// TIA Portal V19 program export: 5 tag tables, 0 data types, 1 data blocks, 10 code blocks (in call order from the OBs), 0 instance data blocks

VAR_GLOBAL   // PLC tag table "Default tag table"
   memSensorType2 AT %MW14 : Int;
   memSensorType1 AT %MW16 : Int;
   Tag_1 AT %T5 : Timer;
END_VAR
VAR_GLOBAL CONSTANT   // user constants
   PANELS_NO : Int := 2;
   LACYCCOM_BUFFER_ELEMENTS_UPPER_LIM : Int := 59;   // Upper limit of request buffer array
   LACYCCOM_WRITE_PARAMETERS_UPPER_LIM : Int := 18;   // Upper limit of write parameters
   LACYCCOM_READ_PARAMETERS_UPPER_LIM : Int := 38;   // Upper limit of read parameters
   LACYCCOM_SILENT_OPERATION_PARAMETERS_UPPER_LIM : Int := 17;   // Upper limit of parameters in LAcycCom_typeDriveSilentOperation
   LACYCCOM_NO_COMMAND : Byte := 16#00;   // No command
   LACYCCOM_READ_COMMAND : Byte := 16#01;   // Read command
   LACYCCOM_WRITE_COMMAND : Byte := 16#02;   // Write command
   LACYCCOM_TYPE_ALARM : SInt := 1;   // Alarm
   LACYCCOM_TYPE_FAULT : SInt := 2;   // Fault
   LACYCCOM_TYPE_SI_MESSAGE : SInt := 3;   // SI message
   LACYCCOM_MESSAGES_UPPER_LIM : Int := 23;   // Upper limit of elements in LAcycCom_typeDriveMessages (fix value)
END_VAR

VAR_GLOBAL   // PLC tag table "tags_IO"
   "866TR2510-S1_Rev" AT %I0.0 : Bool;   // 866TR2510 - Reverse KP-208
   "866TR2510-S1_Fwd" AT %I0.1 : Bool;   // 866TR2510 - Forward KP-208
   "866TR2520-S1_Rev" AT %I0.2 : Bool;   // 866TR2520 - Reverse KP-208
   "866TR2520-S1_Fwd" AT %I0.3 : Bool;   // 866TR2520 - Forward KP-208
   "866TR2530-S1_Rev" AT %I0.4 : Bool;   // 866TR2530 - Reverse KP-208
   "866TR2530-S1_Fwd" AT %I0.5 : Bool;   // 866TR2530 - Forward KP-208
   "866LE2540-S1_Up" AT %I0.6 : Bool;   // 866LE2540 - Cage up
   "866LE2540-S1_Down" AT %I0.7 : Bool;   // 866LE2540 - Cage down
   "866TR2541-S1_Rev" AT %I1.0 : Bool;   // 866TR2541 - Reverse KP-208
   "866TR2541-S1_Fwd" AT %I1.1 : Bool;   // 866TR2541 - Forward KP-208
   "866TR2542-S1_Rev" AT %I1.2 : Bool;   // 866TR2542 - Reverse
   "866TR2542-S1_Fwd" AT %I1.3 : Bool;   // 866TR2542 - Forward
   "866MA2543-S1_In" AT %I1.4 : Bool;   // 866MA2543 - In
   "866MA2543-S1_Out" AT %I1.5 : Bool;   // 866MA2543 - Out
   "866TR2510-GL1" AT %I1.6 : Bool;   // 866TR2510 - Entry photocell
   "866TR2510-GL2" AT %I1.7 : Bool;   // 866TR2510 - Exit photocell
   "866TR2520-GL1" AT %I2.0 : Bool;   // 866TR2520 - Entry photocell
   "866TR2520-GL2" AT %I2.1 : Bool;   // 866TR2520 - Exit photocell
   "866TR2530-GL1" AT %I2.2 : Bool;   // 866TR2530 - Entry photocell
   "866TR2530-GL2" AT %I2.3 : Bool;   // 866TR2530 - Exit photocell
   "2510_KontrollOrd" AT %QW400 : Word;
   "2510_StatusOrd" AT %IW400 : Word;
   "2510_SpeedSP" AT %QW402 : Word;
   "2510_SpeedPV" AT %IW402 : Word;
   "2520_KontrollOrd" AT %QW388 : Word;
   "2520_StatusOrd" AT %IW388 : Word;
   "2520_SpeedSP" AT %QW390 : Word;
   "2520_SpeedPV" AT %IW390 : Word;
   "2530_KontrollOrd" AT %QW376 : Word;
   "2530_StatusOrd" AT %IW376 : Word;
   "2530_SpeedSP" AT %QW378 : Word;
   "2530_SpeedPV" AT %IW378 : Word;
   "2600_KontrollOrd" AT %QW412 : Word;
   "2600_StatusOrd" AT %IW412 : Word;
   "2600_SpeedSP" AT %QW414 : Word;
   "2600_SpeedPV" AT %IW414 : Word;
   "101LT1" AT %IW100 : Word;   // Tank 101 Level transmitter 1
   "101LT2" AT %IW102 : Word;   // Tank 101 Level transmitter 2
   "102LT1" AT %IW104 : Word;   // Tank 102 Level transmitter 1
   "102LT2" AT %IW106 : Word;   // Tank 102 Level transmitter 2
   "101CV1" AT %QW100 : Word;   // Tank 101 Control valve 1
   "101CV2" AT %QW102 : Word;   // Tank 101 Control valve 2
   "102CV1" AT %QW104 : Word;   // Tank 102 Control valve 1
   "102CV2" AT %QW106 : Word;   // Tank 102 Control valve 2
   "101PT1" AT %IW108 : Word;   // Tank 101 Pressure transmitter 1
   "101PT2" AT %IW110 : Word;   // Tank 101 Pressure transmitter 2
   "102PT1" AT %IW112 : Word;   // Tank 102 Pressure transmitter 1
   "102PT2" AT %IW114 : Word;   // Tank 102 Pressure transmitter 2
   "101FT1" AT %IW116 : Word;   // Tank 101 Flow transmitter 1
   "101FT2" AT %IW118 : Word;   // Tank 101 Flow transmitter 2
   "102FT1" AT %IW120 : Word;   // Tank 102 Flow transmitter 1
   "102FT2" AT %IW122 : Word;   // Tank 102 Flow transmitter 2
   "101DV1_GL1" AT %I3.0 : Bool;   // 101DV1 Digital valve open feedback
   "101DV1_GL2" AT %I3.1 : Bool;   // 101DV1 Digital valve closed feedback
   "101DV2_GL1" AT %I3.2 : Bool;   // 101DV2 Digital valve open feedback
   "101DV2_GL2" AT %I3.3 : Bool;   // 101DV2 Digital valve closed feedback
   "101DV1_OPEN" AT %Q0.0 : Bool;
   "101DV2_OPEN" AT %Q0.1 : Bool;
END_VAR

VAR_GLOBAL   // PLC tag table "tags_Omriktare"
   Forward AT %M0.0 : Bool;   // Command
   Backward AT %M0.1 : Bool;   // Command
   Acknowledge AT %M0.2 : Bool;   // Command
   SpeedRequest AT %MW2 : Int;   // Command
   TorqueRequest AT %MW4 : Int;   // Command
   Status AT %MW6 : Word;   // Status
   Speed_CV AT %MW8 : Int;   // Status
   Torque_CV AT %MW10 : Int;   // Status
   Alarm AT %M0.3 : Bool;   // Status
   Alarm_number AT %MW12 : Int;   // Status
END_VAR

VAR_GLOBAL   // PLC tag table "tags_Open Library"
END_VAR
VAR_GLOBAL CONSTANT   // user constants
   "Modes.Auto" : Int := 1;
   "Modes.Manual" : Int := 2;
   "Modes.Independent" : Int := 10;
   "Modes.Stop" : Int := 0;
   "HMI.Status.Stopped" : Int := 0;
   "HMI.Status.Estop" : Int := 1;
   "HMI.Status.Error" : Int := 2;
   "HMI.Status.ForwardWork" : Int := 3;
   "HMI.Status.ReverseHome" : Int := 4;
   "HMI.Status.OnForwardWork" : Int := 5;
   "HMI.Status.OnReverseHome" : Int := 6;
   "IoScaling.S7Analog.Default.iRawMax" : Int := 27648;
   "IoScaling.S7Analog.Default.iRawMin" : Int := 0;
   "IoScaling.S7Analog.Default.bSwapBytes" : Bool := false;
   "IoScaling.S7Analog.+-V/mA.iRawMax" : Int := 27648;
   "IoScaling.S7Analog.+-V/mA.iRawMin" : Int := -27648;
   "IoScaling.S7Analog.Types.Default" : Int := 0;
   "IoScaling.S7Analog.Pt100.iRawMax" : Int := 8500;
   "IoScaling.S7Analog.Pt100.iRawMin" : Int := -2000;
   "IoScaling.S7Analog.Pt100.Climate.iRawMax" : Int := 13000;
   "IoScaling.S7Analog.Pt100.Climate.iRawMin" : Int := -12000;
   "IoScaling.S7Analog.Ni100.iRawMax" : Int := 2500;
   "IoScaling.S7Analog.Ni100.iRawMin" : Int := -600;
   "IoScaling.S7Analog.Ni100.Climate.iRawMax" : Int := 25000;
   "IoScaling.S7Analog.Ni100.Climate.iRawMin" : Int := -6000;
   "IoScaling.S7Analog.Types.+-V/mA" : Int := 1;
   "IoScaling.S7Analog.Types.Pt100" : Int := 2;
   "IoScaling.S7Analog.Types.Pt100.Climate" : Int := 3;
   "IoScaling.S7Analog.Types.Ni100" : Int := 4;
   "IoScaling.S7Analog.Types.Ni100.Climate" : Int := 5;
   "IoScaling.S7Analog.Pt100.rScaledMax" : Real := 850.0;
   "IoScaling.S7Analog.Pt100.rScaledMin" : Real := -200.0;
   "IoScaling.S7Analog.Pt100.Climate.rScaledMax" : Real := 130.0;
   "IoScaling.S7Analog.Pt100.Climate.rScaledMin" : Real := -120.0;
   "IoScaling.S7Analog.Ni100.rScaledMax" : Real := 250.0;
   "IoScaling.S7Analog.Ni100.rScaledMin" : Real := -60.0;
   "IoScaling.S7Analog.Ni100.Climate.rScaledMax" : Real := 250.0;
   "IoScaling.S7Analog.Ni100.Climate.rScaledMin" : Real := -60.0;
   "IoScaling.S7Analog.150Ohms.rScaledMax" : Real := 150.0;
   "IoScaling.S7Analog.150Ohms.rScaledMin" : Real := 0.0;
   "IoScaling.S7Analog.300Ohms.rScaledMax" : Real := 300.0;
   "IoScaling.S7Analog.300Ohms.rScaledMin" : Real := 0.0;
   "IoScaling.S7Analog.600Ohms.rScaledMax" : Real := 600.0;
   "IoScaling.S7Analog.600Ohms.rScaledMin" : Real := 0.0;
   "Estop.MinSetPoint" : Int := 0;
   "Estop.MaxSetPoint" : Int := 1;
   "Estop.HMISetPoint" : Int := 2;
   "Modes.PID.Inactive" : Int := 0;
   "Modes.PID.Pretuning" : Int := 1;
   "Modes.PID.FineTuning" : Int := 2;
   "Modes.PID.AutoMode" : Int := 3;
   "Modes.PID.ManualMode" : Int := 4;
   "HMI.Status.Generic1" : Int := 101;
   "HMI.Status.Generic2" : Int := 102;
   "HMI.Status.Generic3" : Int := 103;
   "HMI.Status.Generic4" : Int := 104;
   "HMI.Status.Generic5" : Int := 105;
   "HMI.Status.GenericNone" : Int := 100;
   "HMI.Status.Generic6" : Int := 106;
   "DataTypes.rMaxReal" : Real := 3.402823e38;
   "DataTypes.rMinReal" : Real := -3.402823e38;
   "DataTypes.iMaxInt" : Int := 32767;
   "DataTypes.iMinInt" : Int := -32768;
   "Handshakes.iSize" : Int := 5;
   "SoftStarter.Types.3RW30" : Int := 30;
   "SoftStarter.Types.3RW40" : Int := 40;
   "Simocode.Types.OverloadRelay" : Int := 0;
   "Simocode.Types.DirectStarter" : Int := 1;
   "Simocode.Types.ReversingStarter" : Int := 2;
   "SoftStarter.HMI.Status.RampDown" : Int := 5;
   "SoftStarter.HMI.Status.On" : Int := 4;
   "SoftStarter.HMI.Status.RampUp" : Int := 3;
   "SoftStarter.HMI.Status.EStop" : Int := 1;
   "SoftStarter.HMI.Status.Off" : Int := 0;
   "SoftStarter.HMI.Status.Error" : Int := 2;
   "FIFO.iQueueSize" : Int := 5;
   "FIFO.iQueueDisabled" : Int := -1;
   "TotalizerTimeUnits.MILLISECONDS" : Int := 0;
   "TotalizerTimeUnits.SECONDS" : Int := 1;
   "TotalizerTimeUnits.MINUTES" : Int := 2;
   "TotalizerTimeUnits.HOURS" : Int := 3;
   "TotalizerTimeUnits.DAYS" : Int := 4;
   "HMI.Status.SimulatedForwardWork" : Int := 7;
   "HMI.Status.SimulatedOnForwardWork" : Int := 9;
   "HMI.Status.SimulatedReverseHome" : Int := 8;
   "HMI.Status.SimulatedOnReverseHome" : Int := 10;
   "Ramp.Continuous" : Int := 0;
   "Ramp.Timed" : Int := 1;
END_VAR

VAR_GLOBAL   // PLC tag table "tags_Testtags"
   V1_Test AT %MD30 : Real;
   V2_Test AT %MD34 : Real;
   T1 AT %M38.0 : Bool;
   T2 AT %M38.1 : Bool;
   T3 AT %M38.2 : Bool;
   T4 AT %M38.3 : Bool;
   T5 AT %M38.4 : Bool;
   TI1 AT %MW40 : Int;
   TI2 AT %MW42 : Int;
   TI3 AT %MW44 : Int;
   TI4 AT %MW46 : Int;
END_VAR

DATA_BLOCK "Interface"   // DB18
{ S7_Optimized_Access := 'TRUE' }
// stored: MemoryReserve 100
   VAR
      LT1_ScaledInput : Real;
      LC1_ControllerOuput : Real;
      LC1_ExtSp : Real := 2.5;
      CV2_ExpSp : Real := 20.0;
      "101CV1_Open" : Bool;
   END_VAR
BEGIN
END_DATA_BLOCK

ORGANIZATION_BLOCK "Drives"   // OB1, FBD, ProgramCycle
TITLE = "Main Program Sweep (Cycle)"
{ S7_Optimized_Access := 'TRUE' }
// stored: SetENOAutomatically false
   VAR_INPUT
      Initial_Call : Bool;   // Initial call of this OB
      Remanence : Bool;   // =True, if remanent data are available
   END_VAR
BEGIN

REGION Network 1: 2510!
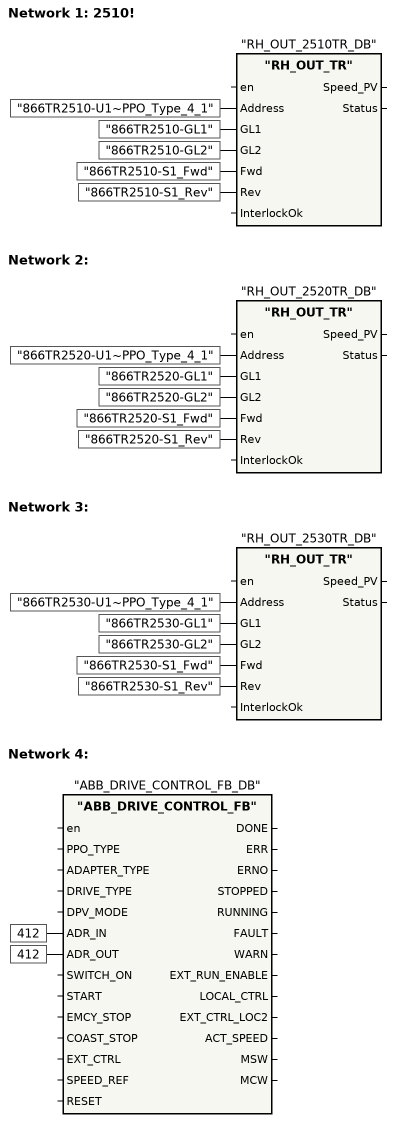
   "RH_OUT_2510TR_DB"(Address := "866TR2510-U1~PPO_Type_4_1",   // "RH_OUT_TR"
                      GL1 := "866TR2510-GL1",
                      GL2 := "866TR2510-GL2",
                      Fwd := "866TR2510-S1_Fwd",
                      Rev := "866TR2510-S1_Rev");
END_REGION

REGION Network 2
   "RH_OUT_2520TR_DB"(Address := "866TR2520-U1~PPO_Type_4_1",   // "RH_OUT_TR"
                      GL1 := "866TR2520-GL1",
                      GL2 := "866TR2520-GL2",
                      Fwd := "866TR2520-S1_Fwd",
                      Rev := "866TR2520-S1_Rev");
END_REGION

REGION Network 3
   "RH_OUT_2530TR_DB"(Address := "866TR2530-U1~PPO_Type_4_1",   // "RH_OUT_TR"
                      GL1 := "866TR2530-GL1",
                      GL2 := "866TR2530-GL2",
                      Fwd := "866TR2530-S1_Fwd",
                      Rev := "866TR2530-S1_Rev");
END_REGION

REGION Network 4
   "ABB_DRIVE_CONTROL_FB_DB"(ADR_IN := 412, ADR_OUT := 412);   // "ABB_DRIVE_CONTROL_FB"
END_REGION
END_ORGANIZATION_BLOCK

FUNCTION_BLOCK "RH_OUT_TR"   // FB1, FBD
{ S7_Optimized_Access := 'TRUE' }
// stored: MemoryReserve 100, SetENOAutomatically false
   VAR_INPUT
      Address : HW_IO;
      GL1 : Bool;
      GL2 : Bool;
      Fwd : Bool;
      Rev : Bool;
      InterlockOk : Bool;
   END_VAR
   VAR_OUTPUT
      Speed_PV : Int;
      Status : Int;
   END_VAR
   VAR
      Frq : "RMP_BIF_FRQ_SPD";   // Device frequency converter control / Laitteen taajuusmuuttajan ohjaus
      Drive { S7_SetPoint := 'True'} : "RMP_FRQ_SPD";
      Control : "RMP_UDT_CONTROL";   // Laitteen ohjaus / Device control
      "Status.Ack" { S7_SetPoint := 'True'} : Bool;
   END_VAR
BEGIN

REGION Network 1: Device fwd request
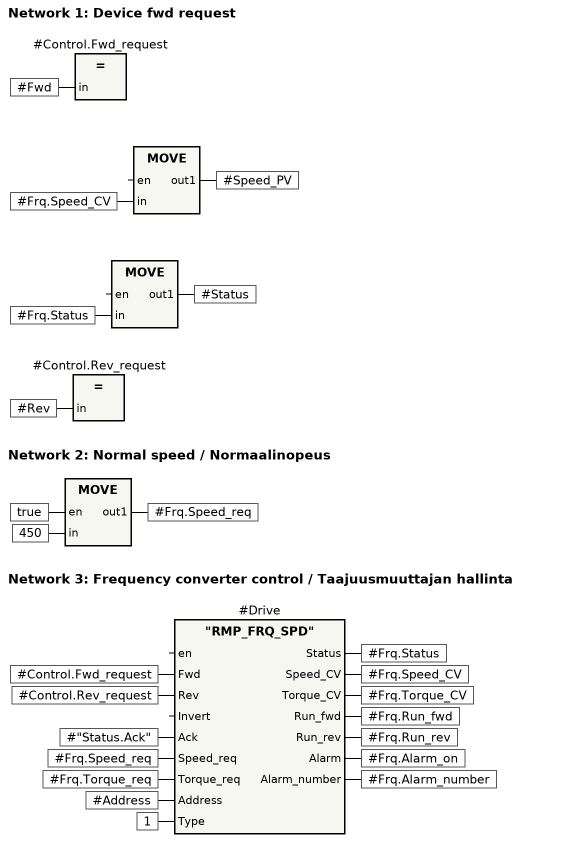
   #Control.Fwd_request := #Fwd;
   #Speed_PV := #Frq.Speed_CV;
   #Status := #Frq.Status;
   #Control.Rev_request := #Rev;
END_REGION

REGION Network 2: Normal speed / Normaalinopeus
   IF true THEN #Frq.Speed_req := 450; END_IF;
END_REGION

REGION Network 3: Frequency converter control / Taajuusmuuttajan hallinta
   #Drive(Fwd := #Control.Fwd_request,   // "RMP_FRQ_SPD"
          Rev := #Control.Rev_request,
          Ack := #"Status.Ack",
          Speed_req := #Frq.Speed_req,
          Torque_req := #Frq.Torque_req,
          Address := #Address,
          "Type" := 1,
          Status => #Frq.Status,
          Speed_CV => #Frq.Speed_CV,
          Torque_CV => #Frq.Torque_CV,
          Run_fwd => #Frq.Run_fwd,
          Run_rev => #Frq.Run_rev,
          Alarm => #Frq.Alarm_on,
          Alarm_number => #Frq.Alarm_number);
END_REGION
END_FUNCTION_BLOCK

FUNCTION_BLOCK "RMP_FRQ_SPD"   // FB11, LAD
TITLE = RMP Sinamics speed & torque control
{ S7_Optimized_Access := 'TRUE' }
AUTHOR : Joni_Lahtonen
FAMILY : Raumaster_Paper
VERSION : 1.0
// This block uses profidrive profile to control siemens frequency converters.
// Use communication profile 352 (6/6) in HW configuration.
// stored: MemoryReserve 100, SetENOAutomatically false
   VAR_INPUT
      Fwd { ExternalAccessible := 'False'; ExternalVisible := 'False'; ExternalWritable := 'False'} : Bool;   // Drive forward request / Eteen käsky
      Rev { ExternalAccessible := 'False'; ExternalVisible := 'False'; ExternalWritable := 'False'} : Bool;   // Drive reverse request / Taakse käsky
      Invert : Bool;   // Invert drive rotation direction / Ajosuunnan muutos
      Ack { ExternalAccessible := 'False'; ExternalVisible := 'False'; ExternalWritable := 'False'} : Bool;   // Drive alarm acknowledge / Häiriönkuittaus
      Speed_req { ExternalAccessible := 'False'; ExternalVisible := 'False'; ExternalWritable := 'False'} : Real;   // Drive speed request 100.0 = 3000rpm / Nopeusohje
      Torque_req { ExternalAccessible := 'False'; ExternalVisible := 'False'; ExternalWritable := 'False'} : Real;   // Drive torque request 100.0 = 100% / Momenttiohje
      Address { ExternalAccessible := 'False'; ExternalVisible := 'False'; ExternalWritable := 'False'} : HW_IO;   // Drive telegram HW address / HW-osoite
      "Type" { ExternalAccessible := 'False'; ExternalVisible := 'False'; ExternalWritable := 'False'} : Bool;   // Drive type 0 = Siemens / 1 = ABB / 0 = Siemens / 1 = ABB
   END_VAR
   VAR_OUTPUT
      Status { ExternalAccessible := 'False'; ExternalVisible := 'False'; ExternalWritable := 'False'} : Word;   // Drive status / Taajuusmuuttajan tilasana
      Speed_CV { ExternalAccessible := 'False'; ExternalVisible := 'False'; ExternalWritable := 'False'} : Real;   // Drive actual speed 100.0 = 3000rpm / Nopeuden oloarvo
      Torque_CV { ExternalAccessible := 'False'; ExternalVisible := 'False'; ExternalWritable := 'False'} : Real;   // Drive actual torgue 100.0 = 100% / Momentin oloarvo
      Run_fwd { ExternalAccessible := 'False'; ExternalVisible := 'False'; ExternalWritable := 'False'} : Bool;   // Drive is running forward / Käy eteen
      Run_rev { ExternalAccessible := 'False'; ExternalVisible := 'False'; ExternalWritable := 'False'} : Bool;   // Drive is running reverse / Käy taakse
      Alarm { ExternalAccessible := 'False'; ExternalVisible := 'False'; ExternalWritable := 'False'} : Bool;   // Drive alarm on / Häiriö päällä
      Alarm_number { ExternalAccessible := 'False'; ExternalVisible := 'False'; ExternalWritable := 'False'} : Int;   // Drive alarm number / Häiriönumero
   END_VAR
   VAR
      Alarm_delay { S7_SetPoint := 'True'} : TON_TIME;
   END_VAR
   VAR_TEMP
      Return_value : Int;
      Siemens : Struct
         In : Struct
            SW : Struct
               Set_point : Bool;   // Setpoint / actual value deviation within the tolerancerange.
               Mst_control_req : Bool;   // The automation system is requested to accept the invertercontrol.
               F_reached : Bool;   // Speed is greater than or equal to the corresponding
               Motor_current_limit : Bool;
               Brake : Bool;
               Motor_overload : Bool;
               CW_CCW_rotation : Bool;
               Converter_overload : Bool;
               Ready_for_on : Bool;   // Power supply switched on; electronics initialized; pulses
               Ready_to_run : Bool;
               Oper_enabled : Bool;   // Motor follows setpoint. See control word 1, bit 3.
               Fault_active : Bool;   // The inverter has a fault. Acknowledge fault using STW1.7.
               OFF2_status : Bool;   // Coast down to standstill is not active.
               OFF3_status : Bool;   // Quick stop is not active.
               Start_lockout : Bool;   // It is only possible to switch on the motor after an OFF1followed by ON.
               Alarm_active : Bool;   // Motor remains switched on; no acknowledgement isnecessary.
            END_STRUCT;
            Speed_CV : Int;
            Data_2 : Int;
            Torque_CV : Int;
            Alarm_nbr : Int;
            Data5 : Int;
         END_STRUCT;
         Out : Struct
            CW : Struct
               Jog_left : Bool;
               Jog_right : Bool;
               Setp_valid : Bool;
               Setp_invert : Bool;
               NC1 : Bool;
               Mop_up : Bool;
               Mop_dn : Bool;
               NC2 : Bool;
               On_Off1 : Bool;   // The motor brakes with the ramp-down time p1121 of theramp-function generator. The inverter switches off the motorat standstill.
               OFF2 : Bool;   // Switch off the motor immediately, the motor then coasts
               OFF3 : Bool;   // Quick stop: The motor brakes with the OFF3 ramp-down
               Oper : Bool;   // Immediately switch-off motor (cancel pulses).
               Cond : Bool;   // The inverter immediately sets its ramp-function generatoroutput to 0.
               Enable_RFG : Bool;   // The output of the ramp-function generator stops at the actualvalue.
               Enable_setpoint : Bool;   // Motor accelerates with the ramp-up time p1120 to thesetpoint
               Ack_fault : Bool;   // Acknowledge fault. If the ON command is still active, theinverter switches to"closing lockout" state.
            END_STRUCT;
            Speed_req : Int;
            Torque_req_p : Int;
            Torque_req_m : Int;
            Data5 : Int;
            Data6 : Int;
         END_STRUCT;
      END_STRUCT;
      ABB : Struct
         In : Struct
            SW : Struct
               At_setpoint : Bool;   // Setpoint / actual value deviation within the tolerancerange. / Actual value equals reference
               Remote : Bool;   // The automation system is requested to accept the invertercontrol. / Drive control location: REMOTE (EXT1 or EXT2)
               Above_limit : Bool;   // Speed is greater than or equal to the corresponding / Actual frequency or speed equals or exceeds supervision limit
               Res_1 : Bool;
               Brake : Bool;   // Brake if parametrized
               Res_3 : Bool;
               Res_4 : Bool;
               FBA_Error : Bool;
               Ready_on : Bool;   // Power supply switched on; electronics initialized; pulses / Ready to switch on
               Ready_run : Bool;   // Ready to operate
               Ready_ref : Bool;   // Motor follows setpoint. See control word 1, bit 3. / Operation enabled
               Tripped : Bool;   // The inverter has a fault. Acknowledge fault using STW1.7. / Fault
               OFF2_status : Bool;   // Coast down to standstill is not active. / OFF 2 inactive
               OFF3_status : Bool;   // Quick stop is not active. / OFF 3 inactive
               Switch_on_inhib : Bool;   // It is only possible to switch on the motor after an OFF1followed by ON. / Switch on inhibited
               Warning : Bool;   // Motor remains switched on; no acknowledgement isnecessary. / Alarm / warning active
            END_STRUCT;
            Speed_CV : Int;
            Data_2 : Int;
            Torque_CV : Int;
            Alarm_nbr : Int;
            Data5 : Int;
         END_STRUCT;
         Out : Struct
            CW : Struct
               Res_1 : Bool;
               Res_2 : Bool;
               Remote_cmd : Bool;
               Ext_ctrl_loc : Bool;
               Res_4 : Bool;
               Res_5 : Bool;
               Res_6 : Bool;
               Res_7 : Bool;
               OFF1_Control : Bool;   // The motor brakes with the ramp-down time p1121 of theramp-function generator. The inverter switches off the motorat standstill.
               OFF2_Control : Bool;   // Switch off the motor immediately, the motor then coasts
               OFF3_Control : Bool;   // Quick stop: The motor brakes with the OFF3 ramp-down
               Inhibit_oper : Bool;   // Immediately switch-off motor (cancel pulses).
               Ramp_out_zero : Bool;   // The inverter immediately sets its ramp-function generatoroutput to 0.
               Ramp_hold : Bool;   // The output of the ramp-function generator stops at the actualvalue.
               Ramp_in_zero : Bool;   // Motor accelerates with the ramp-up time p1120 to thesetpoint
               Reset : Bool;   // Acknowledge fault. If the ON command is still active, theinverter switches to"closing lockout" state.
            END_STRUCT;
            Speed_req : Int;
            Torque_req_p : Int;
            Torque_req_m : Int;
            Data5 : Int;
            Data6 : Int;
         END_STRUCT;
      END_STRUCT;
      Speed_R : Real;
      Torque_R : Real;
      Current_R : Real;
      Speed_req_R : Real;
      Torque_req_R : Real;
      Temp_int : Int;
      Temp_word : Word;
      Error_b : Bool;
      Fwd_req : Bool;
      Setp_invert : Bool;
   END_VAR
BEGIN

REGION Network 1 (SCL): Nopeusohje
   //=========================================================================
   // Raumaster Paper Oy
   // (c)Copyright 2018 All Rights Reserved
   //-----------------------------------------------------------------------------
   // Library: RmpLib
   // Tested with: S7-1516F-3PN/DP V2.1
   //              G120 
   // Engineering: TIA Portal V15
   // Restrictions: 
   // Requirements: S7-1200 / S7-1500
   // Functionality:   This block is made for controlling Siemens drives
   //                  trough Profidrive profile.
   //                  Block uses Siemens telegram 352 6 word in / 6 words out
   //=========================================================================



   IF NOT #Type THEN

       REGION Siemens drive

           //Initialize local variables
           #Siemens.Out.Speed_req := 0;
           #Siemens.Out.Torque_req_p := 0;
           #Temp_word := 0;
           SCATTER(IN := #Temp_word,
                   OUT => #Siemens.Out.CW);

           //Read drive data
           #Return_value := DPRD_DAT(LADDR := #Address, RECORD => #Siemens);

           //Drive status word
           GATHER(IN := #Siemens.In.SW, OUT => #Status);

           #Speed_CV := ABS(INT_TO_REAL(#Siemens.In.Speed_CV) / 16.384);
           #Torque_CV := ABS(INT_TO_REAL(#Siemens.In.Torque_CV) / 16.384);


           //Drive alarm active
           #Alarm_number := #Siemens.In.Alarm_nbr;
           #Alarm_delay(IN := #Siemens.In.SW.Fault_active,
           PT := T#100ms,
           Q => #Alarm);

           //Drive running forward
           #Run_fwd := #Siemens.In.SW.Oper_enabled AND ((NOT #Siemens.In.SW.CW_CCW_rotation AND NOT #Invert) OR (#Siemens.In.SW.CW_CCW_rotation AND #Invert));

           //Drive running reverse
           #Run_rev := #Siemens.In.SW.Oper_enabled AND ((#Siemens.In.SW.CW_CCW_rotation AND NOT #Invert) OR (NOT #Siemens.In.SW.CW_CCW_rotation AND #Invert));

           //Set control bits
           #Siemens.Out.CW.OFF2 := true;
           #Siemens.Out.CW.Oper := true;
           #Siemens.Out.CW.Cond := true;
           #Siemens.Out.CW.Enable_RFG := true;
           #Siemens.Out.CW.Enable_setpoint := true;
           #Siemens.Out.CW.Setp_valid := true;
           #Siemens.Out.CW.OFF3 := true;

           //Drive forward request
           #Fwd_req := (#Fwd OR #Rev) AND #Siemens.In.SW.Ready_for_on AND #Siemens.In.SW.OFF3_status AND NOT #Siemens.In.SW.Fault_active AND NOT #Error_b;

           //Drive forward command
           #Siemens.Out.CW.On_Off1 := #Fwd_req;

           //Drive reverse command
           #Setp_invert := ((#Invert AND NOT #Rev) OR (NOT #Invert AND #Rev)) AND #Fwd_req;

           //Fault ack from drive
           #Siemens.Out.CW.Ack_fault := #Ack;

           //Speed request for drive
           IF #Fwd_req AND NOT #Setp_invert THEN
               #Siemens.Out.Speed_req := REAL_TO_INT(ABS(#Speed_req * 16.384));
           ELSIF #Fwd_req AND #Setp_invert THEN
               #Siemens.Out.Speed_req := - REAL_TO_INT(ABS(#Speed_req * 16.384));
           ELSE
               #Siemens.Out.Speed_req := 0;
           END_IF;


           //Torque request for drive, max positive torque
           #Siemens.Out.Torque_req_p := REAL_TO_INT(#Torque_req * 16.384);
           #Siemens.Out.Torque_req_m := - #Siemens.Out.Torque_req_p;


           //Write drive data
           #Return_value := DPWR_DAT(LADDR := #Address, RECORD := #Siemens.Out);

       END_REGION

   ELSE

       REGION ABB Drive

           //Initialize local variables
           #ABB.Out.Speed_req := 0;
           #ABB.Out.Torque_req_p := 0;
           #Temp_word := 0;
           SCATTER(IN := #Temp_word, OUT => #ABB.Out.CW);

           //Read drive data
           #Return_value := DPRD_DAT(LADDR := #Address, RECORD => #ABB.In);

           //Drive status word
           GATHER(IN := #ABB.In.SW,OUT => #Status);

           #Speed_CV := ABS(INT_TO_REAL(#ABB.In.Speed_CV) / 20.0);
           #Torque_CV := ABS(INT_TO_REAL(#ABB.In.Torque_CV) / 20.0);


           //Drive alarm active
           #Alarm_number := #ABB.In.Alarm_nbr;
           #Alarm_delay(IN := #ABB.In.SW.Tripped, PT := T#200ms, Q => #Alarm);

           //Drive running forward
           #Run_fwd := #ABB.In.SW.Ready_ref AND ((#ABB.In.Speed_CV > 0 AND NOT #Invert) OR (#ABB.In.Speed_CV < 0 AND #Invert));

           //Drive running reverse
           #Run_rev := #ABB.In.SW.Ready_ref AND ((#ABB.In.Speed_CV < 0 AND NOT #Invert) OR (#ABB.In.Speed_CV > 0 AND #Invert));

           //Set control bits
           #ABB.Out.CW.OFF1_Control := #ABB.In.SW.Ready_on;
           #ABB.Out.CW.OFF2_Control := true;
           #ABB.Out.CW.OFF3_Control := true;
           #ABB.Out.CW.Ramp_out_zero := true;
           #ABB.Out.CW.Ramp_hold := true;
           #ABB.Out.CW.Ramp_in_zero := true;
           #ABB.Out.CW.Remote_cmd := true;


           //Drive forward request
           #Fwd_req := (#Fwd OR #Rev) AND NOT #ABB.In.SW.Tripped;// AND #ABB.In.SW.Ready_on AND #ABB.In.SW.OFF3_status

           //Drive forward command
           #ABB.Out.CW.Inhibit_oper := #Fwd_req;

           //Drive reverse command
           #Setp_invert := ((#Invert AND NOT #Rev) OR (NOT #Invert AND #Rev)) AND #Fwd_req;

           //Fault ack from drive
           #ABB.Out.CW.Reset := #Ack;

           //Speed request for drive
           IF #Fwd_req AND NOT #Setp_invert THEN
               #ABB.Out.Speed_req := REAL_TO_INT(ABS(#Speed_req * 20.0));
           ELSIF #Fwd_req AND #Setp_invert THEN
               #ABB.Out.Speed_req := - REAL_TO_INT(ABS(#Speed_req * 20.0));
           ELSE
               #ABB.Out.Speed_req := 0;
           END_IF;

           #ABB.Out.Torque_req_p := REAL_TO_INT(#Torque_req * 20.0);
           #ABB.Out.Torque_req_m := - #ABB.Out.Torque_req_p;

           //Write drive data
           #Return_value := DPWR_DAT(LADDR := #Address, RECORD := #ABB.Out);

       END_REGION
   END_IF;
END_REGION
END_FUNCTION_BLOCK

FUNCTION_BLOCK "ABB_DRIVE_CONTROL_FB"   // FB500, LAD
TITLE = ABB_DRIVE_CONTROL_FB
{ S7_Optimized_Access := 'FALSE' }
AUTHOR : ABB
FAMILY : DRIVES
NAME : ABB
VERSION : 1.3
// stored: SetENOAutomatically false
   VAR_INPUT
      PPO_TYPE : Int;   // PPO-Type: 1,2,3,4,5 or 6; 0 = no fuction
      ADAPTER_TYPE : Int;   // AdapterType:FPBA=1,RPBA=2,FENA=3
      DRIVE_TYPE : Int;   // DriveType: ACS800=1,ACSM1=2,ACS350=3,ACS355=4,ACS550=5,ACS850=6,ACS880=7,ACS580=8,ACSx80=9
      DPV_MODE : Bool;   // FALSE = DP-V0 ; TRUE = DP-V1
      ADR_IN : HW_IO;   // Address of first input byte
      ADR_OUT : HW_IO;   // Address of first output byte
      SWITCH_ON : Bool;   // TRUE = switch on(power on);FALSE = switch off; start power on state machine
      START : Bool;   // TRUE = start enable modulation; FALSE = stop along currently activ stop ramp
      EMCY_STOP : Bool;   // Low active; emergency stop to drive: FALSE = stop by ramp TRUE = no stop
      COAST_STOP : Bool;   // TRUE = coast stop FALSE = normal operation eneble
      EXT_CTRL : Bool;   // External control place 2 EXT2
      SPEED_REF : Int;   // Speed reference value: -20000...20000
   END_VAR
   VAR_OUTPUT
      DONE : Bool;   // Execution finished when output DONE=TRUE
      ERR : Bool;   // Error occured during execution when output ERR=TRUE
      ERNO : Int;   // ErrorCode; see online help SFC14 or SFC15
      STOPPED : Bool;   // The drive has been stopped
      RUNNING : Bool;   // Drive is modulating - following reference
      FAULT : Bool;   // Drive has a fault
      WARN : Bool;   // Drive has a warning
      EXT_RUN_ENABLE : Bool;   // External run enable singal received -> must be set to run
      LOCAL_CTRL : Bool;   // Drive control location LOCAL
      EXT_CTRL_LOC2 : Bool;   // External control location EXT2 selected
      ACT_SPEED : Int;   // Speed actual value: -20000...20000
      MSW : Word;   // Main Status Word
      MCW : Word;   // Actual Main Control Word
   END_VAR
   VAR_IN_OUT
      RESET : Bool;   // Fault acknowled
   END_VAR
   VAR
      Input : Struct
         PPO1 : Struct
            SW : Struct
               AT_SET_POINT : Bool;   // Speed within setpoints
               REMONTE : Bool;   // Profibus control allowed
               ABOVE_LIMIT : Bool;   // Speed / frequency across borders
               EXT_CTRL_LOC : Bool;   // 0=EXT1 1=EXT2 selected
               EXT_RUN_ENABLE : Bool;   // Injury Prevention
               MSV13 : Bool;   // Not in Use
               MSV14 : Bool;   // Not in Use
               COOM_FAULT : Bool;   // Communication Fault Profibus Module CH0
               RDY_ON : Bool;   // Startup finished
               RDY_RUN : Bool;   // Action Completed
               RDY_REF : Bool;   // In Progress
               TRIPPED : Bool;   // Interference
               OFF2_STATE : Bool;   // Freedom freely in the wheels
               OFF3_STATE : Bool;   // Stop as fast as possible
               ON_INHIB : Bool;   // Startup blocked
               ALARM : Bool;   // Alarm
            END_STRUCT;
            Act_Speed : Int;   // Speed
         END_STRUCT;
         PPO2 : Struct
            SW : Struct
               AT_SET_POINT : Bool;   // Speed within setpoints
               REMONTE : Bool;   // Profibus control allowed
               ABOVE_LIMIT : Bool;   // Speed / frequency across borders
               EXT_CTRL_LOC : Bool;   // 0=EXT1 1=EXT2 selected
               EXT_RUN_ENABLE : Bool;   // Injury Prevention
               MSV13 : Bool;   // Not in Use
               MSV14 : Bool;   // Not in Use
               COOM_FAULT : Bool;   // Communication Fault Profibus Module CH0
               RDY_ON : Bool;   // Startup finished
               RDY_RUN : Bool;   // Action Completed
               RDY_REF : Bool;   // In Progress
               TRIPPED : Bool;   // Interference
               OFF2_STATE : Bool;   // Freedom freely in the wheels
               OFF3_STATE : Bool;   // Stop as fast as possible
               ON_INHIB : Bool;   // Startup blocked
               ALARM : Bool;   // Alarm
            END_STRUCT;
            Act_Speed : Int;   // Speed
            PZD_3 : Int;
            PZD_4 : Int;
            PZD_5 : Int;
            PZD_6 : Int;
         END_STRUCT;
         PPO3 : Struct
            SW : Struct
               AT_SET_POINT : Bool;   // Speed within setpoints
               REMONTE : Bool;   // Profibus control allowed
               ABOVE_LIMIT : Bool;   // Speed / frequency across borders
               EXT_CTRL_LOC : Bool;   // 0=EXT1 1=EXT2 selected
               EXT_RUN_ENABLE : Bool;   // Injury Prevention
               MSV13 : Bool;   // Not in Use
               MSV14 : Bool;   // Not in Use
               COOM_FAULT : Bool;   // Communication Fault Profibus Module CH0
               RDY_ON : Bool;   // Startup finished
               RDY_RUN : Bool;   // Action Completed
               RDY_REF : Bool;   // In Progress
               TRIPPED : Bool;   // Interference
               OFF2_STATE : Bool;   // Freedom freely in the wheels
               OFF3_STATE : Bool;   // Stop as fast as possible
               ON_INHIB : Bool;   // Startup blocked
               ALARM : Bool;   // Alarm
            END_STRUCT;
            Act_Speed : Int;   // Speed
         END_STRUCT;
         PPO4 : Struct
            SW : Struct
               AT_SET_POINT : Bool;   // Speed within setpoints
               REMONTE : Bool;   // Profibus control allowed
               ABOVE_LIMIT : Bool;   // Speed / frequency across borders
               EXT_CTRL_LOC : Bool;   // 0=EXT1 1=EXT2 selected
               EXT_RUN_ENABLE : Bool;   // Injury Prevention
               MSV13 : Bool;   // Not in Use
               MSV14 : Bool;   // Not in Use
               COOM_FAULT : Bool;   // Communication Fault Profibus Module CH0
               RDY_ON : Bool;   // Startup finished
               RDY_RUN : Bool;   // Action Completed
               RDY_REF : Bool;   // In Progress
               TRIPPED : Bool;   // Interference
               OFF2_STATE : Bool;   // Freedom freely in the wheels
               OFF3_STATE : Bool;   // Stop as fast as possible
               ON_INHIB : Bool;   // Startup blocked
               ALARM : Bool;   // Alarm
            END_STRUCT;
            Act_Speed : Int;   // Speed
            PZD_3 : Int;
            PZD_4 : Int;
            PZD_5 : Int;
            PZD_6 : Int;
         END_STRUCT;
         PPO5 : Struct
            SW : Struct
               AT_SET_POINT : Bool;   // Speed within setpoints
               REMONTE : Bool;   // Profibus control allowed
               ABOVE_LIMIT : Bool;   // Speed / frequency across borders
               EXT_CTRL_LOC : Bool;   // 0=EXT1 1=EXT2 selected
               EXT_RUN_ENABLE : Bool;   // Injury Prevention
               MSV13 : Bool;   // Not in Use
               MSV14 : Bool;   // Not in Use
               COOM_FAULT : Bool;   // Communication Fault Profibus Module CH0
               RDY_ON : Bool;   // Startup finished
               RDY_RUN : Bool;   // Action Completed
               RDY_REF : Bool;   // In Progress
               TRIPPED : Bool;   // Interference
               OFF2_STATE : Bool;   // Freedom freely in the wheels
               OFF3_STATE : Bool;   // Stop as fast as possible
               ON_INHIB : Bool;   // Startup blocked
               ALARM : Bool;   // Alarm
            END_STRUCT;
            Act_Speed : Int;   // Speed
            PZD_3 : Int;
            PZD_4 : Int;
            PZD_5 : Int;
            PZD_6 : Int;
            PZD_7 : Int;
            PZD_8 : Int;
            PZD_9 : Int;
            PZD_10 : Int;
         END_STRUCT;
         PPO6 : Struct
            SW : Struct
               AT_SET_POINT : Bool;   // Speed within setpoints
               REMONTE : Bool;   // Profibus control allowed
               ABOVE_LIMIT : Bool;   // Speed / frequency across borders
               EXT_CTRL_LOC : Bool;   // 0=EXT1 1=EXT2 selected
               EXT_RUN_ENABLE : Bool;   // Injury Prevention
               MSV13 : Bool;   // Not in Use
               MSV14 : Bool;   // Not in Use
               COOM_FAULT : Bool;   // Communication Fault Profibus Module CH0
               RDY_ON : Bool;   // Startup finished
               RDY_RUN : Bool;   // Action Completed
               RDY_REF : Bool;   // In Progress
               TRIPPED : Bool;   // Interference
               OFF2_STATE : Bool;   // Freedom freely in the wheels
               OFF3_STATE : Bool;   // Stop as fast as possible
               ON_INHIB : Bool;   // Startup blocked
               ALARM : Bool;   // Alarm
            END_STRUCT;
            Act_Speed : Int;   // Speed
            PZD_3 : Int;
            PZD_4 : Int;
            PZD_5 : Int;
            PZD_6 : Int;
            PZD_7 : Int;
            PZD_8 : Int;
            PZD_9 : Int;
            PZD_10 : Int;
         END_STRUCT;
         ACT : Struct
            SW : Struct
               AT_SET_POINT : Bool;   // Speed within setpoints
               REMONTE : Bool;   // Profibus control allowed
               ABOVE_LIMIT : Bool;   // Speed / frequency across borders
               EXT_CTRL_LOC : Bool;   // 0=EXT1 1=EXT2 selected
               EXT_RUN_ENABLE : Bool;   // Injury Prevention
               MSV13 : Bool;   // Not in Use
               MSV14 : Bool;   // Not in Use
               COOM_FAULT : Bool;   // Communication Fault Profibus Module CH0
               RDY_ON : Bool;   // Startup finished
               RDY_RUN : Bool;   // Action Completed
               RDY_REF : Bool;   // In Progress
               TRIPPED : Bool;   // Interference
               OFF2_STATE : Bool;   // Freedom freely in the wheels
               OFF3_STATE : Bool;   // Stop as fast as possible
               ON_INHIB : Bool;   // Startup blocked
               ALARM : Bool;   // Alarm
            END_STRUCT;
            Act_Speed : Int;   // Speed
         END_STRUCT;
      END_STRUCT;
      Output : Struct
         PPO1 : Struct
            CW : Struct
               INCHING_1 : Bool;   // Standard Speed for instruction 1
               INCHING_2 : Bool;   // Standard Speed for instruction 2
               REMONTE_CMD : Bool;   // Profibus control for use
               EXT_CTRL_LOC : Bool;   // 0=EXT1 1=EXT2 selected
               RESERVE_2 : Bool;   // Not in Use
               RESERVE_3 : Bool;   // Not in Use
               RESERVE_4 : Bool;   // Not in Use
               RESERVE_5 : Bool;   // Not in Use
               OFF1 : Bool;   // Start up to readiness
               OFF2 : Bool;   // Free wheel stops
               OFF3 : Bool;   // Emergency stop stop
               INHIBIT_OPREATION : Bool;   // Go to control
               RAMP_OUT_ZERO : Bool;   // Control release
               RAMP_HOLD : Bool;   // Acceleration allowed
               RAMP_IN_ZERO : Bool;   // Speed instruction to zero
               RESET : Bool;   // Fault Reset
            END_STRUCT;
            RefSpeed : Int;
         END_STRUCT;
         PPO2 : Struct
            CW : Struct
               INCHING_1 : Bool;   // Standard Speed for instruction 1
               INCHING_2 : Bool;   // Standard Speed for instruction 2
               REMONTE_CMD : Bool;   // Profibus control for use
               EXT_CTRL_LOC : Bool;   // 0=EXT1 1=EXT2 selected
               RESERVE_2 : Bool;   // Not in Use
               RESERVE_3 : Bool;   // Not in Use
               RESERVE_4 : Bool;   // Not in Use
               RESERVE_5 : Bool;   // Not in Use
               OFF1 : Bool;   // Start up to readiness
               OFF2 : Bool;   // Free wheel stops
               OFF3 : Bool;   // Emergency stop stop
               INHIBIT_OPREATION : Bool;   // Go to control
               RAMP_OUT_ZERO : Bool;   // Control release
               RAMP_HOLD : Bool;   // Acceleration allowed
               RAMP_IN_ZERO : Bool;   // Speed instruction to zero
               RESET : Bool;   // Fault Reset
            END_STRUCT;
            RefSpeed : Int;
            PZD_3 : Int;
            PZD_4 : Int;
            PZD_5 : Int;
            PZD_6 : Int;
         END_STRUCT;
         PPO3 : Struct
            CW : Struct
               INCHING_1 : Bool;   // Standard Speed for instruction 1
               INCHING_2 : Bool;   // Standard Speed for instruction 2
               REMONTE_CMD : Bool;   // Profibus control for use
               EXT_CTRL_LOC : Bool;   // 0=EXT1 1=EXT2 selected
               RESERVE_2 : Bool;   // Not in Use
               RESERVE_3 : Bool;   // Not in Use
               RESERVE_4 : Bool;   // Not in Use
               RESERVE_5 : Bool;   // Not in Use
               OFF1 : Bool;   // Start up to readiness
               OFF2 : Bool;   // Free wheel stops
               OFF3 : Bool;   // Emergency stop stop
               INHIBIT_OPREATION : Bool;   // Go to control
               RAMP_OUT_ZERO : Bool;   // Control release
               RAMP_HOLD : Bool;   // Acceleration allowed
               RAMP_IN_ZERO : Bool;   // Speed instruction to zero
               RESET : Bool;   // Fault Reset
            END_STRUCT;
            RefSpeed : Int;
         END_STRUCT;
         PPO4 : Struct
            CW : Struct
               INCHING_1 : Bool;   // Standard Speed for instruction 1
               INCHING_2 : Bool;   // Standard Speed for instruction 2
               REMONTE_CMD : Bool;   // Profibus control for use
               EXT_CTRL_LOC : Bool;   // 0=EXT1 1=EXT2 selected
               RESERVE_2 : Bool;   // Not in Use
               RESERVE_3 : Bool;   // Not in Use
               RESERVE_4 : Bool;   // Not in Use
               RESERVE_5 : Bool;   // Not in Use
               OFF1 : Bool;   // Start up to readiness
               OFF2 : Bool;   // Free wheel stops
               OFF3 : Bool;   // Emergency stop stop
               INHIBIT_OPREATION : Bool;   // Go to control
               RAMP_OUT_ZERO : Bool;   // Control release
               RAMP_HOLD : Bool;   // Acceleration allowed
               RAMP_IN_ZERO : Bool;   // Speed instruction to zero
               RESET : Bool;   // Fault Reset
            END_STRUCT;
            RefSpeed : Int;
            PZD_3 : Int;
            PZD_4 : Int;
            PZD_5 : Int;
            PZD_6 : Int;
         END_STRUCT;
         PPO5 : Struct
            CW : Struct
               INCHING_1 : Bool;   // Standard Speed for instruction 1
               INCHING_2 : Bool;   // Standard Speed for instruction 2
               REMONTE_CMD : Bool;   // Profibus control for use
               EXT_CTRL_LOC : Bool;   // 0=EXT1 1=EXT2 selected
               RESERVE_2 : Bool;   // Not in Use
               RESERVE_3 : Bool;   // Not in Use
               RESERVE_4 : Bool;   // Not in Use
               RESERVE_5 : Bool;   // Not in Use
               OFF1 : Bool;   // Start up to readiness
               OFF2 : Bool;   // Free wheel stops
               OFF3 : Bool;   // Emergency stop stop
               INHIBIT_OPREATION : Bool;   // Go to control
               RAMP_OUT_ZERO : Bool;   // Control release
               RAMP_HOLD : Bool;   // Acceleration allowed
               RAMP_IN_ZERO : Bool;   // Speed instruction to zero
               RESET : Bool;   // Fault Reset
            END_STRUCT;
            RefSpeed : Int;
            PZD_3 : Int;
            PZD_4 : Int;
            PZD_5 : Int;
            PZD_6 : Int;
            PZD_7 : Int;
            PZD_8 : Int;
            PZD_9 : Int;
            PZD_10 : Int;
         END_STRUCT;
         PPO6 : Struct
            CW : Struct
               INCHING_1 : Bool;   // Standard Speed for instruction 1
               INCHING_2 : Bool;   // Standard Speed for instruction 2
               REMONTE_CMD : Bool;   // Profibus control for use
               EXT_CTRL_LOC : Bool;   // 0=EXT1 1=EXT2 selected
               RESERVE_2 : Bool;   // Not in Use
               RESERVE_3 : Bool;   // Not in Use
               RESERVE_4 : Bool;   // Not in Use
               RESERVE_5 : Bool;   // Not in Use
               OFF1 : Bool;   // Start up to readiness
               OFF2 : Bool;   // Free wheel stops
               OFF3 : Bool;   // Emergency stop stop
               INHIBIT_OPREATION : Bool;   // Go to control
               RAMP_OUT_ZERO : Bool;   // Control release
               RAMP_HOLD : Bool;   // Acceleration allowed
               RAMP_IN_ZERO : Bool;   // Speed instruction to zero
               RESET : Bool;   // Fault Reset
            END_STRUCT;
            RefSpeed : Int;
            PZD_3 : Int;
            PZD_4 : Int;
            PZD_5 : Int;
            PZD_6 : Int;
            PZD_7 : Int;
            PZD_8 : Int;
            PZD_9 : Int;
            PZD_10 : Int;
         END_STRUCT;
         ACT : Struct
            CW : Struct
               INCHING_1 : Bool;   // Standard Speed for instruction 1
               INCHING_2 : Bool;   // Standard Speed for instruction 2
               REMONTE_CMD : Bool;   // Profibus control for use
               EXT_CTRL_LOC : Bool;   // 0=EXT1 1=EXT2 selected
               RESERVE_2 : Bool;   // Not in Use
               RESERVE_3 : Bool;   // Not in Use
               RESERVE_4 : Bool;   // Not in Use
               RESERVE_5 : Bool;   // Not in Use
               OFF1 : Bool;   // Start up to readiness
               OFF2 : Bool;   // Free wheel stops
               OFF3 : Bool;   // Emergency stop stop
               INHIBIT_OPREATION : Bool;   // Go to control
               RAMP_OUT_ZERO : Bool;   // Control release
               RAMP_HOLD : Bool;   // Acceleration allowed
               RAMP_IN_ZERO : Bool;   // Speed instruction to zero
               RESET : Bool;   // Fault Reset
            END_STRUCT;
            RefSpeed : Int;
         END_STRUCT;
      END_STRUCT;
      PARA_INTERNAL_DPV0 : Struct
         Done : Bool;
         Err : Bool;
         Busy : Bool;
         Read_FB : Bool;
         Write_FB : Bool;
         Time_out : Bool;
         Read_request : Bool;
         Write_Request : Bool;
         Parameter_access : Bool;
         Para_9 : Bool;
         Para_10 : Bool;
         Para_11 : Bool;
         Para_12 : Bool;
         Para_13 : Bool;
         Para_14 : Bool;
         Para_15 : Bool;
         Para_16 : Bool;
         Para_17 : Bool;
         Para_18 : Bool;
         Para_19 : Bool;
         Para_20 : Bool;
         Para_21 : Bool;
         Para_22 : Bool;
         Para_23 : Bool;
         Para_24 : Bool;
         Para_25 : Bool;
         Para_26 : Bool;
         Para_27 : Bool;
         Para_28 : Bool;
         Para_29 : Bool;
         Para_30 : Bool;
         PDV_MODE : Bool;   // DP-V0 = 0 (false) / DP-V1 = 1 (true)
         RESPONCE_LABEL : Int;
         PARA_NUM_OUT : Int;
         PARA_NUM_INDEX_OUT : Int;
         PARA_ERR_NRO : Word;
         PARA_VALUE_OUT : DInt;
         ADDRESS_IN : Word;
         ADDRESS_OUT : Word;
         Master_to_Slave : Struct
            ID : Word;   // Request Label bits 4-7 Parameter number bits 0-2
            IND : Word;   // Parameter number index bits 0-15
            VALUE : DWord;   // Parameter values
         END_STRUCT;
         Slave_to_Master : Struct
            ID : Word;   // Request Label bits 4-7 Parameter number bits 0-2
            IND : Word;   // Parameter number index bits 0-15
            VALUE : DWord;   // Parameter values
         END_STRUCT;
         PPO_TYPE : Int;   // PPO-Type: 1,2,3,4,5 or 6; 0 = no fuction
         ADAPTER_TYPE : Int;   // AdapterType:FPBA=1,RPBA=2,FENA=3
         DRIVE_TYPE : Int;
      END_STRUCT;
      PARA_INTERNAL_DPV1 : Struct
         Request : Struct
            Reference : Byte;
            ID : Byte;   // 1 read / 2 change
            Axis : Byte;
            NoOfParameters : Byte;
            Attribute : Byte;
            NoOfElements : Byte;
            ParameterIndex : Word;
            Subindex : Word;
            Format : Byte;
            NumberOfValues : Byte;
            Value : DWord;
         END_STRUCT;
         Responce : Struct
            Reference : Byte;
            ID : Byte;
            Axis : Byte;
            NoOfParametrs : Byte;
            Format : Byte;
            NoOfValues : Byte;
            Value : DWord;
         END_STRUCT;
         Request_DONE : Bool;
         Request_BUSY : Bool;
         Request_ERROR : Bool;
         Request_STATUS : DWord;
         Responce_VALID : Bool;
         Responce_BUSY : Bool;
         Responce_ERROR : Bool;
         Responce_STATUS : DWord;
         Responce_LEN : UInt;
      END_STRUCT;
      INTERNAL_PZD : Struct
         IN : Struct
            PZD2 : Int;
            PZD3 : Int;
            PZD4 : Int;
            PZD5 : Int;
            PZD6 : Int;
            PZD7 : Int;
            PZD8 : Int;
            PZD9 : Int;
            PZD10 : Int;
         END_STRUCT;
         OUT : Struct
            PZD3 : Int;
            PZD4 : Int;
            PZD5 : Int;
            PZD6 : Int;
            PZD7 : Int;
            PZD8 : Int;
            PZD9 : Int;
            PZD10 : Int;
         END_STRUCT;
         SCALED : Struct
            PZD2 : Real;
            PZD3 : Real;
            PZD4 : Real;
            PZD5 : Real;
            PZD6 : Real;
            PZD7 : Real;
            PZD8 : Real;
            PZD9 : Real;
            PZD10 : Real;
         END_STRUCT;
         SCALE : Struct
            PZD2_SCALE : Real;
            PZD3_SCALE : Real;
            PZD4_SCALE : Real;
            PZD5_SCALE : Real;
            PZD6_SCALE : Real;
            PZD7_SCALE : Real;
            PZD8_SCALE : Real;
            PZD9_SCALE : Real;
            PZD10_SCALE : Real;
         END_STRUCT;
      END_STRUCT;
      DPV1_WRITE { S7_SetPoint := 'True'} : WRREC;
      DPV1_READ { S7_SetPoint := 'True'} : WRREC;
      DP1_RESPONCE { S7_SetPoint := 'True'} : RDREC;
      INPUT_ADDRESS : Word;
      OUTPUT_ADDRESS : Word;
      RET_VAL_INPUT : Int;
      RET_VAL_OUTPUT : Int;
      DONE_ON : Bool;
      ParameterErr : Bool;
      ERROR : Bool;
      READ_FAULT : Bool;
      SWITCH_ON_FP : Bool;
      POWER_STATE : Int;
      ALLWAYS_ON : Bool;
      ALLWAYS_OFF : Bool;
      POWER_ON : Bool;
      RESET_POWER_ON : Bool;
      PARA_TIME_OUT { S7_SetPoint := 'True'} : TON_TIME;
      INTERNA_ERR : Int;
      POWER_RESET_FB : Bool;
      PARA_NUM : DInt;
      PARA_VALUE : DInt;
      PARA_INTERNAL_DPV1_16bit : Struct
         Request : Struct
            Reference : Byte;
            ID : Byte;   // 1 read / 2 change
            Axis : Byte;
            NoOfParameters : Byte;
            Attribute : Byte := B#16#10;
            NoOfElements : Byte;
            ParameterIndex : Word;
            Subindex : Word;
            Format : Byte;
            NumberOfValues : Byte;
            Value : Word;
         END_STRUCT;
         Responce : Struct
            Reference : Byte;
            ID : Byte;
            Axis : Byte;
            NoOfParametrs : Byte;
            Format : Byte;
            NoOfValues : Byte;
            Value : DWord;
         END_STRUCT;
         Request_DONE : Bool;
         Request_BUSY : Bool;
         Request_ERROR : Bool;
         Request_STATUS : DWord;
         Responce_VALID : Bool;
         Responce_BUSY : Bool;
         Responce_ERROR : Bool;
         Responce_STATUS : DWord;
         Responce_LEN : Int;
      END_STRUCT;
      Drive_Type_Dummy : Bool;
      Drive_Type_Dummy2 : Bool;
      Response_Format_Dummy : Int;
      Format_Check : Bool;
      Format_Check_1 : Bool;
      Request_Sent_32bit : Bool;
      Request_Sent_16bit : Bool;
      Request_Sent_16bit_1 : Bool;
      RESTART : Bool;
      RESTART_EMG : Bool;
      POWER_RESET_FB_1 : Bool;
   END_VAR
   VAR_TEMP
      PARA_READ_ERR : Int;
      TEMP0 : Time;
      IN_ADDRESS_DW : Word;
      OUT_ADDRESS_DW : Word;
      dummy : Bool;
      MSW_Temp : Struct
         SW : Struct
            AT_SET_POINT : Bool;   // Nopeus asetusarvojen sisällä
            REMONTE : Bool;   // Profibuss ohjaus sallittu
            ABOVE_LIMIT : Bool;   // Nopeus / taajuus yli rajojen
            EXT_CTRL_LOC : Bool;   // 0=EXT1 1=EXT2 selected
            EXT_RUN_ENABLE : Bool;   // Vahinkokäynnistyksen esto
            MSV13 : Bool;   // Ei käytössä
            MSV14 : Bool;   // Ei käytössä
            COOM_FAULT : Bool;   // Kommunikointivika profibus moduuli CH0
            RDY_ON : Bool;   // Käynnistys valmis
            RDY_RUN : Bool;   // Toiminta valmis
            RDY_REF : Bool;   // Käynnissä
            TRIPPED : Bool;   // Häiriö
            OFF2_STATE : Bool;   // Pysäytys vapaasti pyörien
            OFF3_STATE : Bool;   // Pysäytys hahdollisimman nopeasti
            ON_INHIB : Bool;   // Käynnistys estetty
            ALARM : Bool;   // Hälytys
         END_STRUCT;
      END_STRUCT;
      MSW_Conv AT MSW_Temp : Word;
      MCW_Temp : Struct
         CW : Struct
            INCHING_1 : Bool;   // Vakio nopeus ohje 1 käyttöön
            INCHING_2 : Bool;   // Vakio nopeus ohje 2 käyttöön
            REMONTE_CMD : Bool;   // Profibuss ohjaus käyttöön
            EXT_CTRL_LOC : Bool;   // 0=EXT1 1=EXT2 selected
            RESERVE_2 : Bool;   // Ei käytössä
            RESERVE_3 : Bool;   // Ei käytössä
            RESERVE_4 : Bool;   // Ei käytössä
            RESERVE_5 : Bool;   // Ei käytössä
            OFF1 : Bool;   // Käynnistys valmiuteen
            OFF2 : Bool;   // Vapaastipyörien seis
            OFF3 : Bool;   // Hätä-seis pysäytys
            INHIBIT_OPREATION : Bool;   // Käyntiin ohjaus
            RAMP_OUT_ZERO : Bool;   // Ohjauksen vapautus
            RAMP_HOLD : Bool;   // Kiihdytys sallittu
            RAMP_IN_ZERO : Bool;   // Nopeus ohje nollaan
            RESET : Bool;   // Häiriön kuittaus
         END_STRUCT;
      END_STRUCT;
      MCW_Conv AT MCW_Temp : Word;
      "ReadRequest Sent" : Bool;
      PowerState_Temp : Int;
   END_VAR
   VAR_TEMP   // added for the SCL form of the ladder/FBD networks
      _w1 : Bool;
      _w2 : Bool;
      _w3 : Bool;
      _w4 : Bool;
   END_VAR
BEGIN

REGION Network 1: Set init values
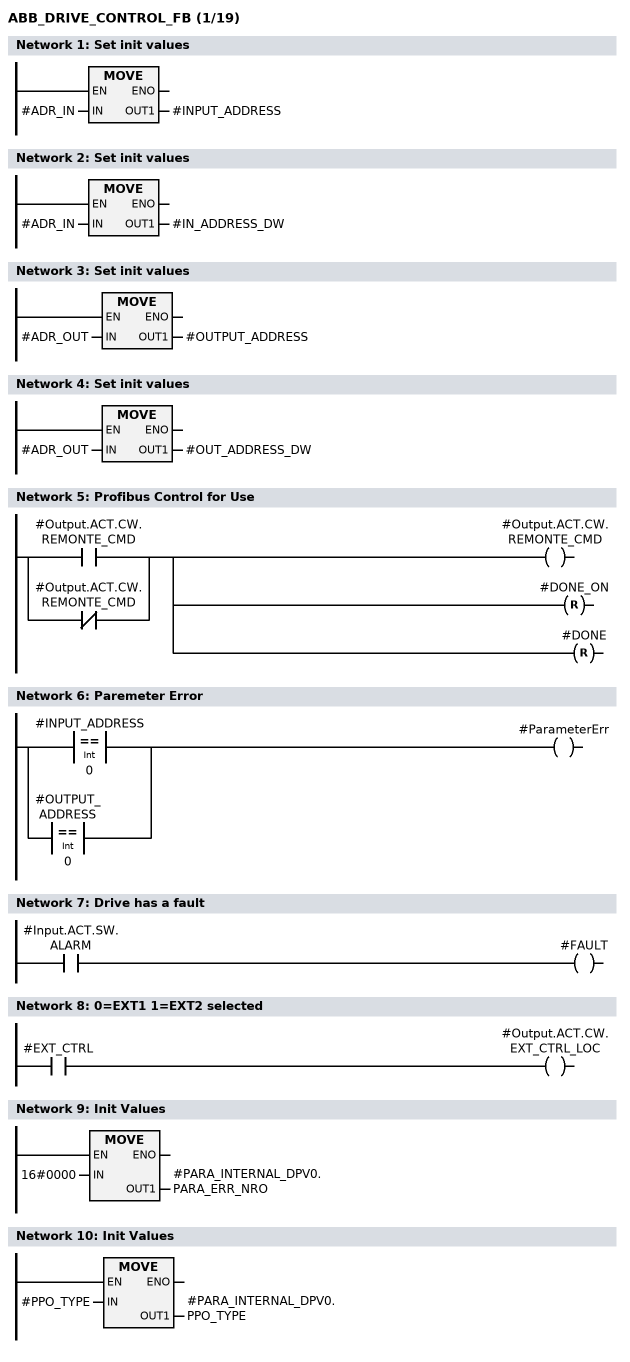
   RUNG wire#powerrail
      { S7_GenerateENO := "TRUE" } Move(in := #ADR_IN, out1 => #INPUT_ADDRESS)
   END_RUNG
   // the same network as SCL:
   #INPUT_ADDRESS := #ADR_IN;
END_REGION

REGION Network 2: Set init values
   RUNG wire#powerrail
      { S7_GenerateENO := "TRUE" } Move(in := #ADR_IN, out1 => #IN_ADDRESS_DW)
   END_RUNG
   // the same network as SCL:
   #IN_ADDRESS_DW := #ADR_IN;
END_REGION

REGION Network 3: Set init values
   RUNG wire#powerrail
      { S7_GenerateENO := "TRUE" } Move(in := #ADR_OUT, out1 => #OUTPUT_ADDRESS)
   END_RUNG
   // the same network as SCL:
   #OUTPUT_ADDRESS := #ADR_OUT;
END_REGION

REGION Network 4: Set init values
   RUNG wire#powerrail
      { S7_GenerateENO := "TRUE" } Move(in := #ADR_OUT, out1 => #OUT_ADDRESS_DW)
   END_RUNG
   // the same network as SCL:
   #OUT_ADDRESS_DW := #ADR_OUT;
END_REGION

REGION Network 5: Profibus Control for Use
   RUNG wire#powerrail
      Contact( #Output.ACT.CW.REMONTE_CMD )
      wire#w1
      Coil( #Output.ACT.CW.REMONTE_CMD )
   END_RUNG
   RUNG wire#powerrail
      I_Contact( #Output.ACT.CW.REMONTE_CMD )
   END_RUNG wire#w1
   RUNG wire#w1
      R_Coil( #DONE_ON )
   END_RUNG
   RUNG wire#w1
      R_Coil( #DONE )
   END_RUNG
   // the same network as SCL:
   #Output.ACT.CW.REMONTE_CMD := #Output.ACT.CW.REMONTE_CMD OR NOT #Output.ACT.CW.REMONTE_CMD;
   IF #Output.ACT.CW.REMONTE_CMD THEN
       #DONE_ON := FALSE;
       #DONE := FALSE;
   END_IF;
END_REGION

REGION Network 6: Paremeter Error
   RUNG wire#powerrail
      { S7_Templates := "SrcType := Int" } EQ_Contact(in1 := #INPUT_ADDRESS, in2 := 0)
      wire#w1
      Coil( #ParameterErr )
   END_RUNG
   RUNG wire#powerrail
      { S7_Templates := "SrcType := Int" } EQ_Contact(in1 := #OUTPUT_ADDRESS, in2 := 0)
   END_RUNG wire#w1
   // the same network as SCL:
   #ParameterErr := (#INPUT_ADDRESS = 0) OR (#OUTPUT_ADDRESS = 0);
END_REGION

REGION Network 7: Drive has a fault
   RUNG wire#powerrail
      Contact( #Input.ACT.SW.ALARM )
      Coil( #FAULT )
   END_RUNG
   // the same network as SCL:
   #FAULT := #Input.ACT.SW.ALARM;
END_REGION

REGION Network 8: 0=EXT1 1=EXT2 selected
   RUNG wire#powerrail
      Contact( #EXT_CTRL )
      Coil( #Output.ACT.CW.EXT_CTRL_LOC )
   END_RUNG
   // the same network as SCL:
   #Output.ACT.CW.EXT_CTRL_LOC := #EXT_CTRL;
END_REGION

REGION Network 9: Init Values
   RUNG wire#powerrail
      { S7_GenerateENO := "TRUE" } Move(in := 16#0000, out1 => #PARA_INTERNAL_DPV0.PARA_ERR_NRO)
   END_RUNG
   // the same network as SCL:
   #PARA_INTERNAL_DPV0.PARA_ERR_NRO := 16#0000;
END_REGION

REGION Network 10: Init Values
   RUNG wire#powerrail
      { S7_GenerateENO := "TRUE" } Move(in := #PPO_TYPE, out1 => #PARA_INTERNAL_DPV0.PPO_TYPE)
   END_RUNG
   // the same network as SCL:
   #PARA_INTERNAL_DPV0.PPO_TYPE := #PPO_TYPE;
END_REGION

REGION Network 11: Init Values
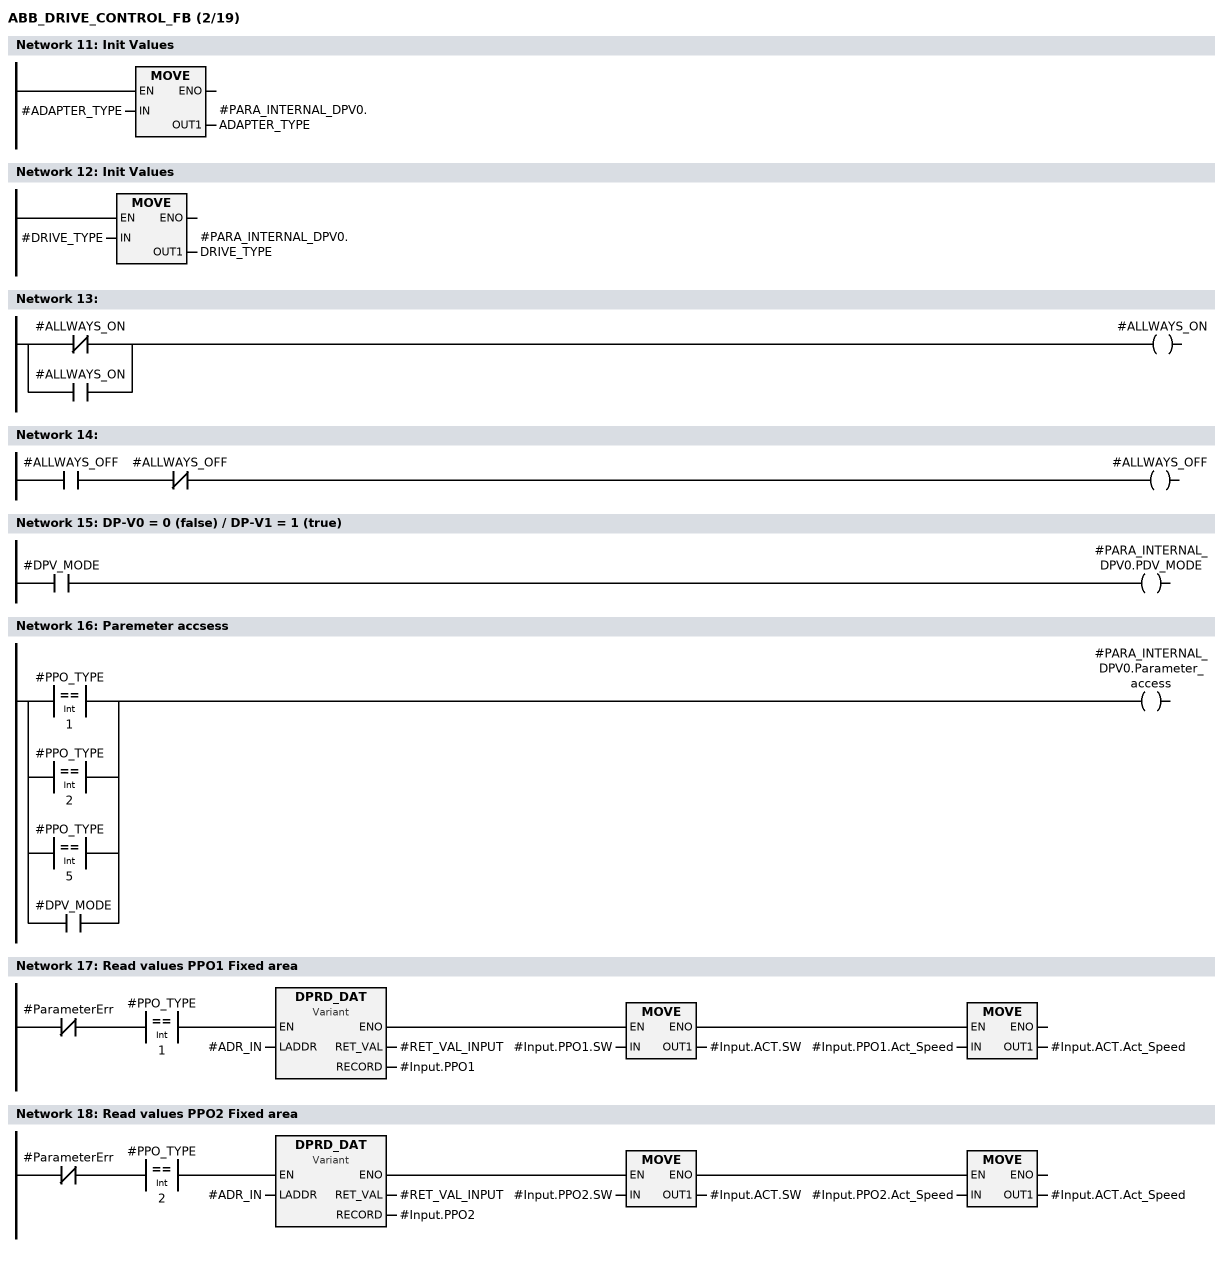
   RUNG wire#powerrail
      { S7_GenerateENO := "TRUE" } Move(in := #ADAPTER_TYPE, out1 => #PARA_INTERNAL_DPV0.ADAPTER_TYPE)
   END_RUNG
   // the same network as SCL:
   #PARA_INTERNAL_DPV0.ADAPTER_TYPE := #ADAPTER_TYPE;
END_REGION

REGION Network 12: Init Values
   RUNG wire#powerrail
      { S7_GenerateENO := "TRUE" } Move(in := #DRIVE_TYPE, out1 => #PARA_INTERNAL_DPV0.DRIVE_TYPE)
   END_RUNG
   // the same network as SCL:
   #PARA_INTERNAL_DPV0.DRIVE_TYPE := #DRIVE_TYPE;
END_REGION

REGION Network 13
   RUNG wire#powerrail
      I_Contact( #ALLWAYS_ON )
      wire#w1
      Coil( #ALLWAYS_ON )
   END_RUNG
   RUNG wire#powerrail
      Contact( #ALLWAYS_ON )
   END_RUNG wire#w1
   // the same network as SCL:
   #ALLWAYS_ON := NOT #ALLWAYS_ON OR #ALLWAYS_ON;
END_REGION

REGION Network 14
   RUNG wire#powerrail
      Contact( #ALLWAYS_OFF )
      I_Contact( #ALLWAYS_OFF )
      Coil( #ALLWAYS_OFF )
   END_RUNG
   // the same network as SCL:
   #ALLWAYS_OFF := #ALLWAYS_OFF AND NOT #ALLWAYS_OFF;
END_REGION

REGION Network 15: DP-V0 = 0 (false) / DP-V1 = 1 (true)
   RUNG wire#powerrail
      Contact( #DPV_MODE )
      Coil( #PARA_INTERNAL_DPV0.PDV_MODE )
   END_RUNG
   // the same network as SCL:
   #PARA_INTERNAL_DPV0.PDV_MODE := #DPV_MODE;
END_REGION

REGION Network 16: Paremeter accsess
   RUNG wire#powerrail
      { S7_Templates := "SrcType := Int" } EQ_Contact(in1 := #PPO_TYPE, in2 := 1)
      wire#w1
      Coil( #PARA_INTERNAL_DPV0.Parameter_access )
   END_RUNG
   RUNG wire#powerrail
      { S7_Templates := "SrcType := Int" } EQ_Contact(in1 := #PPO_TYPE, in2 := 2)
   END_RUNG wire#w1
   RUNG wire#powerrail
      { S7_Templates := "SrcType := Int" } EQ_Contact(in1 := #PPO_TYPE, in2 := 5)
   END_RUNG wire#w1
   RUNG wire#powerrail
      Contact( #DPV_MODE )
   END_RUNG wire#w1
   // the same network as SCL:
   #PARA_INTERNAL_DPV0.Parameter_access := (#PPO_TYPE = 1) OR (#PPO_TYPE = 2) OR (#PPO_TYPE = 5) OR #DPV_MODE;
END_REGION

REGION Network 17: Read values PPO1 Fixed area
   RUNG wire#powerrail
      I_Contact( #ParameterErr )
      { S7_Templates := "SrcType := Int" } EQ_Contact(in1 := #PPO_TYPE, in2 := 1)
      { S7_Templates := "[ptr_type := Variant, laddr_type := HW_IO]" } DPRD_DAT(LADDR := #ADR_IN, RET_VAL => #RET_VAL_INPUT, RECORD => #Input.PPO1)
      { S7_GenerateENO := "TRUE" } Move(in := #Input.PPO1.SW, out1 => #Input.ACT.SW)
      { S7_GenerateENO := "TRUE" } Move(in := #Input.PPO1.Act_Speed, out1 => #Input.ACT.Act_Speed)
   END_RUNG
   // the same network as SCL:
   // ENO of a box is taken as its EN; it also drops when the box reports an error
   #RET_VAL_INPUT := DPRD_DAT(EN := NOT #ParameterErr AND (#PPO_TYPE = 1),
                           LADDR := #ADR_IN,
                           RECORD => #Input.PPO1,
                           ENO => #_w1);
   IF #_w1 THEN
       #Input.ACT.SW := #Input.PPO1.SW;
       #Input.ACT.Act_Speed := #Input.PPO1.Act_Speed;
   END_IF;
END_REGION

REGION Network 18: Read values PPO2 Fixed area
   RUNG wire#powerrail
      I_Contact( #ParameterErr )
      { S7_Templates := "SrcType := Int" } EQ_Contact(in1 := #PPO_TYPE, in2 := 2)
      { S7_Templates := "[ptr_type := Variant, laddr_type := HW_IO]" } DPRD_DAT(LADDR := #ADR_IN, RET_VAL => #RET_VAL_INPUT, RECORD => #Input.PPO2)
      { S7_GenerateENO := "TRUE" } Move(in := #Input.PPO2.SW, out1 => #Input.ACT.SW)
      { S7_GenerateENO := "TRUE" } Move(in := #Input.PPO2.Act_Speed, out1 => #Input.ACT.Act_Speed)
   END_RUNG
   // the same network as SCL:
   // ENO of a box is taken as its EN; it also drops when the box reports an error
   #RET_VAL_INPUT := DPRD_DAT(EN := NOT #ParameterErr AND (#PPO_TYPE = 2),
                           LADDR := #ADR_IN,
                           RECORD => #Input.PPO2,
                           ENO => #_w1);
   IF #_w1 THEN
       #Input.ACT.SW := #Input.PPO2.SW;
       #Input.ACT.Act_Speed := #Input.PPO2.Act_Speed;
   END_IF;
END_REGION

REGION Network 19: Move PPO2 Process data area
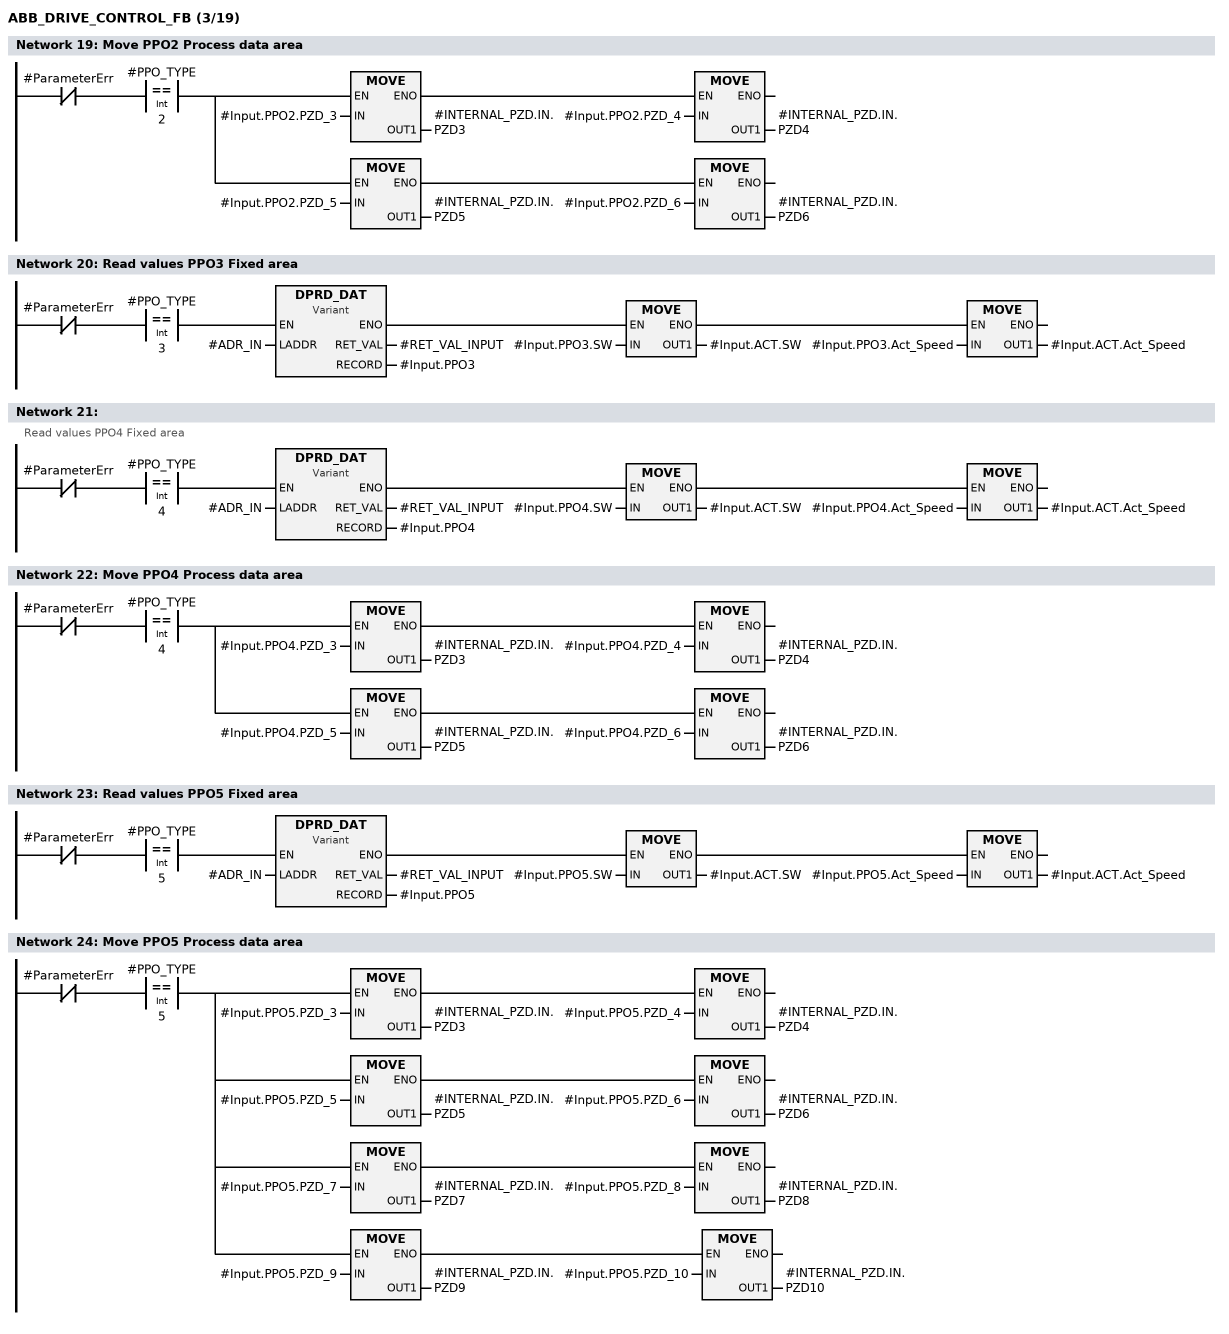
   RUNG wire#powerrail
      I_Contact( #ParameterErr )
      { S7_Templates := "SrcType := Int" } EQ_Contact(in1 := #PPO_TYPE, in2 := 2)
      wire#w1
      { S7_GenerateENO := "TRUE" } Move(in := #Input.PPO2.PZD_3, out1 => #INTERNAL_PZD.IN.PZD3)
      { S7_GenerateENO := "TRUE" } Move(in := #Input.PPO2.PZD_4, out1 => #INTERNAL_PZD.IN.PZD4)
   END_RUNG
   RUNG wire#w1
      { S7_GenerateENO := "TRUE" } Move(in := #Input.PPO2.PZD_5, out1 => #INTERNAL_PZD.IN.PZD5)
      { S7_GenerateENO := "TRUE" } Move(in := #Input.PPO2.PZD_6, out1 => #INTERNAL_PZD.IN.PZD6)
   END_RUNG
   // the same network as SCL:
   // ENO of a box is taken as its EN; it also drops when the box reports an error
   IF NOT #ParameterErr AND (#PPO_TYPE = 2) THEN
       #INTERNAL_PZD.IN.PZD3 := #Input.PPO2.PZD_3;
       #INTERNAL_PZD.IN.PZD4 := #Input.PPO2.PZD_4;
       #INTERNAL_PZD.IN.PZD5 := #Input.PPO2.PZD_5;
       #INTERNAL_PZD.IN.PZD6 := #Input.PPO2.PZD_6;
   END_IF;
END_REGION

REGION Network 20: Read values PPO3 Fixed area
   RUNG wire#powerrail
      I_Contact( #ParameterErr )
      { S7_Templates := "SrcType := Int" } EQ_Contact(in1 := #PPO_TYPE, in2 := 3)
      { S7_Templates := "[ptr_type := Variant, laddr_type := HW_IO]" } DPRD_DAT(LADDR := #ADR_IN, RET_VAL => #RET_VAL_INPUT, RECORD => #Input.PPO3)
      { S7_GenerateENO := "TRUE" } Move(in := #Input.PPO3.SW, out1 => #Input.ACT.SW)
      { S7_GenerateENO := "TRUE" } Move(in := #Input.PPO3.Act_Speed, out1 => #Input.ACT.Act_Speed)
   END_RUNG
   // the same network as SCL:
   // ENO of a box is taken as its EN; it also drops when the box reports an error
   #RET_VAL_INPUT := DPRD_DAT(EN := NOT #ParameterErr AND (#PPO_TYPE = 3),
                           LADDR := #ADR_IN,
                           RECORD => #Input.PPO3,
                           ENO => #_w1);
   IF #_w1 THEN
       #Input.ACT.SW := #Input.PPO3.SW;
       #Input.ACT.Act_Speed := #Input.PPO3.Act_Speed;
   END_IF;
END_REGION

REGION Network 21
   // Read values PPO4 Fixed area
   RUNG wire#powerrail
      I_Contact( #ParameterErr )
      { S7_Templates := "SrcType := Int" } EQ_Contact(in1 := #PPO_TYPE, in2 := 4)
      { S7_Templates := "[ptr_type := Variant, laddr_type := HW_IO]" } DPRD_DAT(LADDR := #ADR_IN, RET_VAL => #RET_VAL_INPUT, RECORD => #Input.PPO4)
      { S7_GenerateENO := "TRUE" } Move(in := #Input.PPO4.SW, out1 => #Input.ACT.SW)
      { S7_GenerateENO := "TRUE" } Move(in := #Input.PPO4.Act_Speed, out1 => #Input.ACT.Act_Speed)
   END_RUNG
   // the same network as SCL:
   // ENO of a box is taken as its EN; it also drops when the box reports an error
   #RET_VAL_INPUT := DPRD_DAT(EN := NOT #ParameterErr AND (#PPO_TYPE = 4),
                           LADDR := #ADR_IN,
                           RECORD => #Input.PPO4,
                           ENO => #_w1);
   IF #_w1 THEN
       #Input.ACT.SW := #Input.PPO4.SW;
       #Input.ACT.Act_Speed := #Input.PPO4.Act_Speed;
   END_IF;
END_REGION

REGION Network 22: Move PPO4 Process data area
   RUNG wire#powerrail
      I_Contact( #ParameterErr )
      { S7_Templates := "SrcType := Int" } EQ_Contact(in1 := #PPO_TYPE, in2 := 4)
      wire#w1
      { S7_GenerateENO := "TRUE" } Move(in := #Input.PPO4.PZD_3, out1 => #INTERNAL_PZD.IN.PZD3)
      { S7_GenerateENO := "TRUE" } Move(in := #Input.PPO4.PZD_4, out1 => #INTERNAL_PZD.IN.PZD4)
   END_RUNG
   RUNG wire#w1
      { S7_GenerateENO := "TRUE" } Move(in := #Input.PPO4.PZD_5, out1 => #INTERNAL_PZD.IN.PZD5)
      { S7_GenerateENO := "TRUE" } Move(in := #Input.PPO4.PZD_6, out1 => #INTERNAL_PZD.IN.PZD6)
   END_RUNG
   // the same network as SCL:
   // ENO of a box is taken as its EN; it also drops when the box reports an error
   IF NOT #ParameterErr AND (#PPO_TYPE = 4) THEN
       #INTERNAL_PZD.IN.PZD3 := #Input.PPO4.PZD_3;
       #INTERNAL_PZD.IN.PZD4 := #Input.PPO4.PZD_4;
       #INTERNAL_PZD.IN.PZD5 := #Input.PPO4.PZD_5;
       #INTERNAL_PZD.IN.PZD6 := #Input.PPO4.PZD_6;
   END_IF;
END_REGION

REGION Network 23: Read values PPO5 Fixed area
   RUNG wire#powerrail
      I_Contact( #ParameterErr )
      { S7_Templates := "SrcType := Int" } EQ_Contact(in1 := #PPO_TYPE, in2 := 5)
      { S7_Templates := "[ptr_type := Variant, laddr_type := HW_IO]" } DPRD_DAT(LADDR := #ADR_IN, RET_VAL => #RET_VAL_INPUT, RECORD => #Input.PPO5)
      { S7_GenerateENO := "TRUE" } Move(in := #Input.PPO5.SW, out1 => #Input.ACT.SW)
      { S7_GenerateENO := "TRUE" } Move(in := #Input.PPO5.Act_Speed, out1 => #Input.ACT.Act_Speed)
   END_RUNG
   // the same network as SCL:
   // ENO of a box is taken as its EN; it also drops when the box reports an error
   #RET_VAL_INPUT := DPRD_DAT(EN := NOT #ParameterErr AND (#PPO_TYPE = 5),
                           LADDR := #ADR_IN,
                           RECORD => #Input.PPO5,
                           ENO => #_w1);
   IF #_w1 THEN
       #Input.ACT.SW := #Input.PPO5.SW;
       #Input.ACT.Act_Speed := #Input.PPO5.Act_Speed;
   END_IF;
END_REGION

REGION Network 24: Move PPO5 Process data area
   RUNG wire#powerrail
      I_Contact( #ParameterErr )
      { S7_Templates := "SrcType := Int" } EQ_Contact(in1 := #PPO_TYPE, in2 := 5)
      wire#w1
      { S7_GenerateENO := "TRUE" } Move(in := #Input.PPO5.PZD_3, out1 => #INTERNAL_PZD.IN.PZD3)
      { S7_GenerateENO := "TRUE" } Move(in := #Input.PPO5.PZD_4, out1 => #INTERNAL_PZD.IN.PZD4)
   END_RUNG
   RUNG wire#w1
      { S7_GenerateENO := "TRUE" } Move(in := #Input.PPO5.PZD_5, out1 => #INTERNAL_PZD.IN.PZD5)
      { S7_GenerateENO := "TRUE" } Move(in := #Input.PPO5.PZD_6, out1 => #INTERNAL_PZD.IN.PZD6)
   END_RUNG
   RUNG wire#w1
      { S7_GenerateENO := "TRUE" } Move(in := #Input.PPO5.PZD_7, out1 => #INTERNAL_PZD.IN.PZD7)
      { S7_GenerateENO := "TRUE" } Move(in := #Input.PPO5.PZD_8, out1 => #INTERNAL_PZD.IN.PZD8)
   END_RUNG
   RUNG wire#w1
      { S7_GenerateENO := "TRUE" } Move(in := #Input.PPO5.PZD_9, out1 => #INTERNAL_PZD.IN.PZD9)
      { S7_GenerateENO := "TRUE" } Move(in := #Input.PPO5.PZD_10, out1 => #INTERNAL_PZD.IN.PZD10)
   END_RUNG
   // the same network as SCL:
   // ENO of a box is taken as its EN; it also drops when the box reports an error
   IF NOT #ParameterErr AND (#PPO_TYPE = 5) THEN
       #INTERNAL_PZD.IN.PZD3 := #Input.PPO5.PZD_3;
       #INTERNAL_PZD.IN.PZD4 := #Input.PPO5.PZD_4;
       #INTERNAL_PZD.IN.PZD5 := #Input.PPO5.PZD_5;
       #INTERNAL_PZD.IN.PZD6 := #Input.PPO5.PZD_6;
       #INTERNAL_PZD.IN.PZD7 := #Input.PPO5.PZD_7;
       #INTERNAL_PZD.IN.PZD8 := #Input.PPO5.PZD_8;
       #INTERNAL_PZD.IN.PZD9 := #Input.PPO5.PZD_9;
       #INTERNAL_PZD.IN.PZD10 := #Input.PPO5.PZD_10;
   END_IF;
END_REGION

REGION Network 25: Read values PPO6 Fixed area
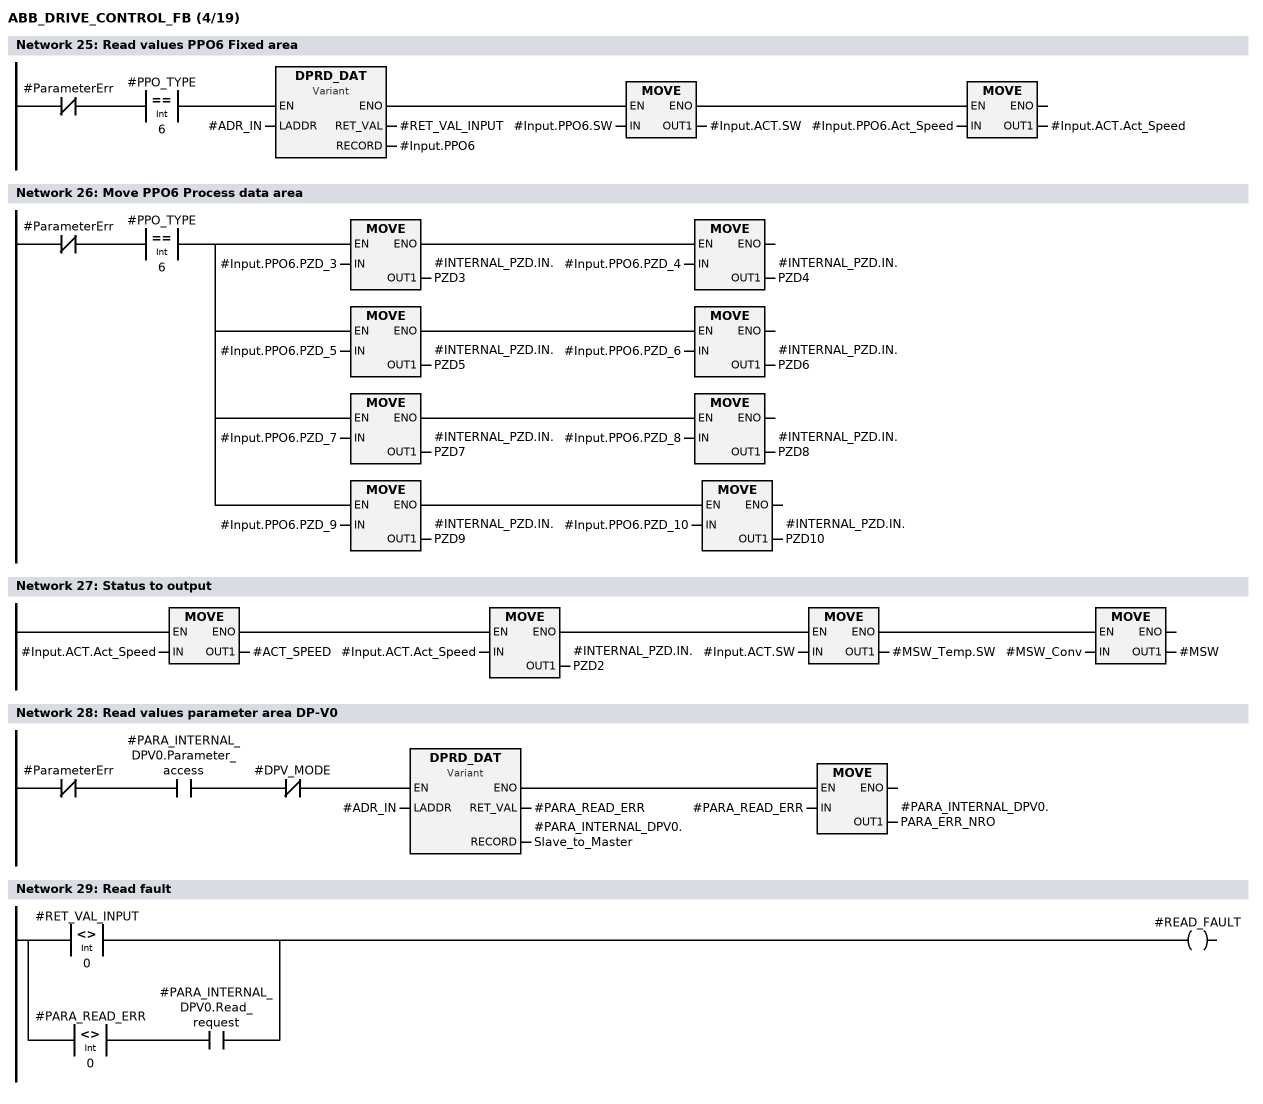
   RUNG wire#powerrail
      I_Contact( #ParameterErr )
      { S7_Templates := "SrcType := Int" } EQ_Contact(in1 := #PPO_TYPE, in2 := 6)
      { S7_Templates := "[ptr_type := Variant, laddr_type := HW_IO]" } DPRD_DAT(LADDR := #ADR_IN, RET_VAL => #RET_VAL_INPUT, RECORD => #Input.PPO6)
      { S7_GenerateENO := "TRUE" } Move(in := #Input.PPO6.SW, out1 => #Input.ACT.SW)
      { S7_GenerateENO := "TRUE" } Move(in := #Input.PPO6.Act_Speed, out1 => #Input.ACT.Act_Speed)
   END_RUNG
   // the same network as SCL:
   // ENO of a box is taken as its EN; it also drops when the box reports an error
   #RET_VAL_INPUT := DPRD_DAT(EN := NOT #ParameterErr AND (#PPO_TYPE = 6),
                           LADDR := #ADR_IN,
                           RECORD => #Input.PPO6,
                           ENO => #_w1);
   IF #_w1 THEN
       #Input.ACT.SW := #Input.PPO6.SW;
       #Input.ACT.Act_Speed := #Input.PPO6.Act_Speed;
   END_IF;
END_REGION

REGION Network 26: Move PPO6 Process data area
   RUNG wire#powerrail
      I_Contact( #ParameterErr )
      { S7_Templates := "SrcType := Int" } EQ_Contact(in1 := #PPO_TYPE, in2 := 6)
      wire#w1
      { S7_GenerateENO := "TRUE" } Move(in := #Input.PPO6.PZD_3, out1 => #INTERNAL_PZD.IN.PZD3)
      { S7_GenerateENO := "TRUE" } Move(in := #Input.PPO6.PZD_4, out1 => #INTERNAL_PZD.IN.PZD4)
   END_RUNG
   RUNG wire#w1
      { S7_GenerateENO := "TRUE" } Move(in := #Input.PPO6.PZD_5, out1 => #INTERNAL_PZD.IN.PZD5)
      { S7_GenerateENO := "TRUE" } Move(in := #Input.PPO6.PZD_6, out1 => #INTERNAL_PZD.IN.PZD6)
   END_RUNG
   RUNG wire#w1
      { S7_GenerateENO := "TRUE" } Move(in := #Input.PPO6.PZD_7, out1 => #INTERNAL_PZD.IN.PZD7)
      { S7_GenerateENO := "TRUE" } Move(in := #Input.PPO6.PZD_8, out1 => #INTERNAL_PZD.IN.PZD8)
   END_RUNG
   RUNG wire#w1
      { S7_GenerateENO := "TRUE" } Move(in := #Input.PPO6.PZD_9, out1 => #INTERNAL_PZD.IN.PZD9)
      { S7_GenerateENO := "TRUE" } Move(in := #Input.PPO6.PZD_10, out1 => #INTERNAL_PZD.IN.PZD10)
   END_RUNG
   // the same network as SCL:
   // ENO of a box is taken as its EN; it also drops when the box reports an error
   IF NOT #ParameterErr AND (#PPO_TYPE = 6) THEN
       #INTERNAL_PZD.IN.PZD3 := #Input.PPO6.PZD_3;
       #INTERNAL_PZD.IN.PZD4 := #Input.PPO6.PZD_4;
       #INTERNAL_PZD.IN.PZD5 := #Input.PPO6.PZD_5;
       #INTERNAL_PZD.IN.PZD6 := #Input.PPO6.PZD_6;
       #INTERNAL_PZD.IN.PZD7 := #Input.PPO6.PZD_7;
       #INTERNAL_PZD.IN.PZD8 := #Input.PPO6.PZD_8;
       #INTERNAL_PZD.IN.PZD9 := #Input.PPO6.PZD_9;
       #INTERNAL_PZD.IN.PZD10 := #Input.PPO6.PZD_10;
   END_IF;
END_REGION

REGION Network 27: Status to output
   RUNG wire#powerrail
      { S7_GenerateENO := "TRUE" } Move(in := #Input.ACT.Act_Speed, out1 => #ACT_SPEED)
      { S7_GenerateENO := "TRUE" } Move(in := #Input.ACT.Act_Speed, out1 => #INTERNAL_PZD.IN.PZD2)
      { S7_GenerateENO := "TRUE" } Move(in := #Input.ACT.SW, out1 => #MSW_Temp.SW)
      { S7_GenerateENO := "TRUE" } Move(in := #MSW_Conv, out1 => #MSW)
   END_RUNG
   // the same network as SCL:
   // ENO of a box is taken as its EN; it also drops when the box reports an error
   #ACT_SPEED := #Input.ACT.Act_Speed;
   #INTERNAL_PZD.IN.PZD2 := #Input.ACT.Act_Speed;
   #MSW_Temp.SW := #Input.ACT.SW;
   #MSW := #MSW_Conv;
END_REGION

REGION Network 28: Read values parameter area DP-V0
   RUNG wire#powerrail
      I_Contact( #ParameterErr )
      Contact( #PARA_INTERNAL_DPV0.Parameter_access )
      I_Contact( #DPV_MODE )
      { S7_Templates := "[ptr_type := Variant, laddr_type := HW_IO]" } DPRD_DAT(LADDR := #ADR_IN, RET_VAL => #PARA_READ_ERR, RECORD => #PARA_INTERNAL_DPV0.Slave_to_Master)
      { S7_GenerateENO := "TRUE" } Move(in := #PARA_READ_ERR, out1 => #PARA_INTERNAL_DPV0.PARA_ERR_NRO)
   END_RUNG
   // the same network as SCL:
   #PARA_READ_ERR := DPRD_DAT(EN := NOT #ParameterErr AND #PARA_INTERNAL_DPV0.Parameter_access AND NOT #DPV_MODE,
                           LADDR := #ADR_IN,
                           RECORD => #PARA_INTERNAL_DPV0.Slave_to_Master,
                           ENO => #_w1);
   IF #_w1 THEN #PARA_INTERNAL_DPV0.PARA_ERR_NRO := #PARA_READ_ERR; END_IF;
END_REGION

REGION Network 29: Read fault
   RUNG wire#powerrail
      { S7_Templates := "SrcType := Int" } NE_Contact(in1 := #RET_VAL_INPUT, in2 := 0)
      wire#w1
      Coil( #READ_FAULT )
   END_RUNG
   RUNG wire#powerrail
      { S7_Templates := "SrcType := Int" } NE_Contact(in1 := #PARA_READ_ERR, in2 := 0)
      Contact( #PARA_INTERNAL_DPV0.Read_request )
   END_RUNG wire#w1
   // the same network as SCL:
   #READ_FAULT := (#RET_VAL_INPUT <> 0) OR ((#PARA_READ_ERR <> 0) AND #PARA_INTERNAL_DPV0.Read_request);
END_REGION

REGION Network 30: Power on
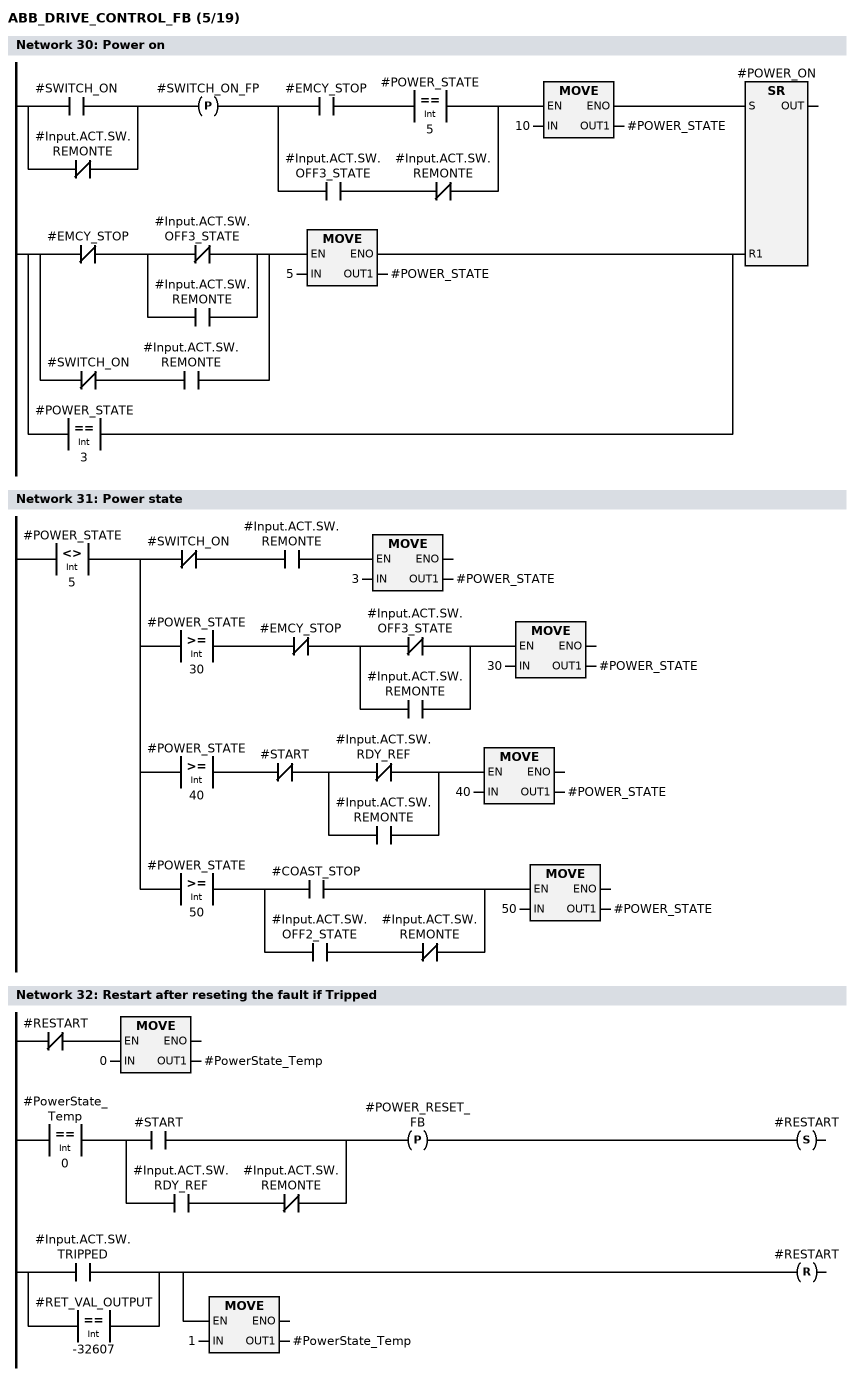
   RUNG wire#powerrail
      Contact( #SWITCH_ON )
      wire#w1
      P_Trig( #SWITCH_ON_FP )
      wire#w2
      Contact( #EMCY_STOP )
      { S7_Templates := "SrcType := Int" } EQ_Contact(in1 := #POWER_STATE, in2 := 5)
      wire#w3
      { S7_GenerateENO := "TRUE" } Move(in := 10, out1 => #POWER_STATE)
      S_SR(operand := #POWER_ON, r1 := wire#w6)
   END_RUNG
   RUNG wire#powerrail
      I_Contact( #Input.ACT.SW.REMONTE )
   END_RUNG wire#w1
   RUNG wire#w2
      Contact( #Input.ACT.SW.OFF3_STATE )
      I_Contact( #Input.ACT.SW.REMONTE )
   END_RUNG wire#w3
   RUNG wire#powerrail
      I_Contact( #EMCY_STOP )
      wire#w4
      I_Contact( #Input.ACT.SW.OFF3_STATE )
      wire#w5
      { S7_GenerateENO := "TRUE" } Move(in := 5, out1 => #POWER_STATE)
   END_RUNG wire#w6
   RUNG wire#w4
      Contact( #Input.ACT.SW.REMONTE )
   END_RUNG wire#w5
   RUNG wire#powerrail
      I_Contact( #SWITCH_ON )
      Contact( #Input.ACT.SW.REMONTE )
   END_RUNG wire#w5
   RUNG wire#powerrail
      { S7_Templates := "SrcType := Int" } EQ_Contact(in1 := #POWER_STATE, in2 := 3)
   END_RUNG wire#w6
   // the same network as SCL:
   // ENO of a box is taken as its EN; it also drops when the box reports an error
   #_w1 := #SWITCH_ON OR NOT #Input.ACT.SW.REMONTE;
   #_w2 := #_w1 AND NOT #SWITCH_ON_FP;   // rising edge
   #SWITCH_ON_FP := #_w1;
   #_w3 := #_w2 AND ((#EMCY_STOP AND (#POWER_STATE = 5)) OR (#Input.ACT.SW.OFF3_STATE AND NOT #Input.ACT.SW.REMONTE));
   IF #_w3 THEN #POWER_STATE := 10; END_IF;
   #_w4 := (NOT #EMCY_STOP AND (NOT #Input.ACT.SW.OFF3_STATE OR #Input.ACT.SW.REMONTE)) OR (NOT #SWITCH_ON AND #Input.ACT.SW.REMONTE);
   IF #_w4 THEN #POWER_STATE := 5; END_IF;
   IF #_w3 THEN
       #POWER_ON := TRUE;   // SR flip-flop
   END_IF;
   IF #_w4 OR (#POWER_STATE = 3) THEN #POWER_ON := FALSE; END_IF;
END_REGION

REGION Network 31: Power state
   RUNG wire#powerrail
      { S7_Templates := "SrcType := Int" } NE_Contact(in1 := #POWER_STATE, in2 := 5)
      wire#w1
      I_Contact( #SWITCH_ON )
      Contact( #Input.ACT.SW.REMONTE )
      { S7_GenerateENO := "TRUE" } Move(in := 3, out1 => #POWER_STATE)
   END_RUNG
   RUNG wire#w1
      { S7_Templates := "SrcType := Int" } GE_Contact(in1 := #POWER_STATE, in2 := 30)
      I_Contact( #EMCY_STOP )
      wire#w2
      I_Contact( #Input.ACT.SW.OFF3_STATE )
      wire#w3
      { S7_GenerateENO := "TRUE" } Move(in := 30, out1 => #POWER_STATE)
   END_RUNG
   RUNG wire#w2
      Contact( #Input.ACT.SW.REMONTE )
   END_RUNG wire#w3
   RUNG wire#w1
      { S7_Templates := "SrcType := Int" } GE_Contact(in1 := #POWER_STATE, in2 := 40)
      I_Contact( #START )
      wire#w4
      I_Contact( #Input.ACT.SW.RDY_REF )
      wire#w5
      { S7_GenerateENO := "TRUE" } Move(in := 40, out1 => #POWER_STATE)
   END_RUNG
   RUNG wire#w4
      Contact( #Input.ACT.SW.REMONTE )
   END_RUNG wire#w5
   RUNG wire#w1
      { S7_Templates := "SrcType := Int" } GE_Contact(in1 := #POWER_STATE, in2 := 50)
      wire#w6
      Contact( #COAST_STOP )
      wire#w7
      { S7_GenerateENO := "TRUE" } Move(in := 50, out1 => #POWER_STATE)
   END_RUNG
   RUNG wire#w6
      Contact( #Input.ACT.SW.OFF2_STATE )
      I_Contact( #Input.ACT.SW.REMONTE )
   END_RUNG wire#w7
   // the same network as SCL:
   #_w1 := #POWER_STATE <> 5;
   IF #_w1 AND NOT #SWITCH_ON AND #Input.ACT.SW.REMONTE THEN #POWER_STATE := 3; END_IF;
   IF #_w1 AND (#POWER_STATE >= 30) AND NOT #EMCY_STOP AND (NOT #Input.ACT.SW.OFF3_STATE OR #Input.ACT.SW.REMONTE) THEN
       #POWER_STATE := 30;
   END_IF;
   IF #_w1 AND (#POWER_STATE >= 40) AND NOT #START AND (NOT #Input.ACT.SW.RDY_REF OR #Input.ACT.SW.REMONTE) THEN
       #POWER_STATE := 40;
   END_IF;
   IF #_w1 AND (#POWER_STATE >= 50) AND (#COAST_STOP OR (#Input.ACT.SW.OFF2_STATE AND NOT #Input.ACT.SW.REMONTE)) THEN
       #POWER_STATE := 50;
   END_IF;
END_REGION

REGION Network 32: Restart after reseting the fault if Tripped
   RUNG wire#powerrail
      I_Contact( #RESTART )
      Move(in := 0, out1 => #PowerState_Temp)
   END_RUNG
   RUNG wire#powerrail
      { S7_Templates := "SrcType := Int" } EQ_Contact(in1 := #PowerState_Temp, in2 := 0)
      wire#w1
      Contact( #START )
      wire#w2
      P_Trig( #POWER_RESET_FB )
      S_Coil( #RESTART )
   END_RUNG
   RUNG wire#w1
      Contact( #Input.ACT.SW.RDY_REF )
      I_Contact( #Input.ACT.SW.REMONTE )
   END_RUNG wire#w2
   RUNG wire#powerrail
      Contact( #Input.ACT.SW.TRIPPED )
      wire#w3
      R_Coil( #RESTART )
   END_RUNG
   RUNG wire#powerrail
      { S7_Templates := "SrcType := Int" } EQ_Contact(in1 := #RET_VAL_OUTPUT, in2 := -32607)
   END_RUNG wire#w3
   RUNG wire#w3
      Move(in := 1, out1 => #PowerState_Temp)
   END_RUNG
   // the same network as SCL:
   IF NOT #RESTART THEN #PowerState_Temp := 0; END_IF;
   #_w1 := (#PowerState_Temp = 0) AND (#START OR (#Input.ACT.SW.RDY_REF AND NOT #Input.ACT.SW.REMONTE));
   #_w2 := #_w1 AND NOT #POWER_RESET_FB;   // rising edge
   #POWER_RESET_FB := #_w1;
   IF #_w2 THEN #RESTART := TRUE; END_IF;
   IF #Input.ACT.SW.TRIPPED OR (#RET_VAL_OUTPUT = (-32607)) THEN
       #RESTART := FALSE;
       #PowerState_Temp := 1;
   END_IF;
END_REGION

REGION Network 33: Restart after reseting the fault if EmergencyStop exist
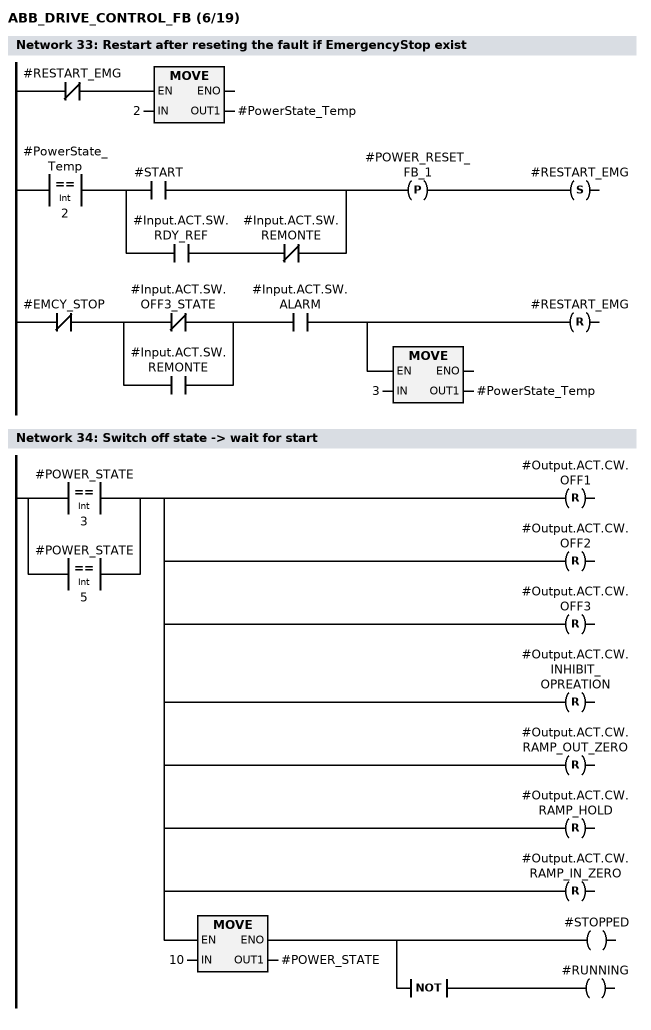
   RUNG wire#powerrail
      I_Contact( #RESTART_EMG )
      Move(in := 2, out1 => #PowerState_Temp)
   END_RUNG
   RUNG wire#powerrail
      { S7_Templates := "SrcType := Int" } EQ_Contact(in1 := #PowerState_Temp, in2 := 2)
      wire#w1
      Contact( #START )
      wire#w2
      P_Trig( #POWER_RESET_FB_1 )
      S_Coil( #RESTART_EMG )
   END_RUNG
   RUNG wire#w1
      Contact( #Input.ACT.SW.RDY_REF )
      I_Contact( #Input.ACT.SW.REMONTE )
   END_RUNG wire#w2
   RUNG wire#powerrail
      I_Contact( #EMCY_STOP )
      wire#w3
      I_Contact( #Input.ACT.SW.OFF3_STATE )
      wire#w4
      Contact( #Input.ACT.SW.ALARM )
      wire#w5
      R_Coil( #RESTART_EMG )
   END_RUNG
   RUNG wire#w3
      Contact( #Input.ACT.SW.REMONTE )
   END_RUNG wire#w4
   RUNG wire#w5
      Move(in := 3, out1 => #PowerState_Temp)
   END_RUNG
   // the same network as SCL:
   IF NOT #RESTART_EMG THEN #PowerState_Temp := 2; END_IF;
   #_w1 := (#PowerState_Temp = 2) AND (#START OR (#Input.ACT.SW.RDY_REF AND NOT #Input.ACT.SW.REMONTE));
   #_w2 := #_w1 AND NOT #POWER_RESET_FB_1;   // rising edge
   #POWER_RESET_FB_1 := #_w1;
   IF #_w2 THEN #RESTART_EMG := TRUE; END_IF;
   IF NOT #EMCY_STOP AND (NOT #Input.ACT.SW.OFF3_STATE OR #Input.ACT.SW.REMONTE) AND #Input.ACT.SW.ALARM THEN
       #RESTART_EMG := FALSE;
       #PowerState_Temp := 3;
   END_IF;
END_REGION

REGION Network 34: Switch off state -> wait for start
   RUNG wire#powerrail
      { S7_Templates := "SrcType := Int" } EQ_Contact(in1 := #POWER_STATE, in2 := 3)
      wire#w1
      R_Coil( #Output.ACT.CW.OFF1 )
   END_RUNG
   RUNG wire#powerrail
      { S7_Templates := "SrcType := Int" } EQ_Contact(in1 := #POWER_STATE, in2 := 5)
   END_RUNG wire#w1
   RUNG wire#w1
      R_Coil( #Output.ACT.CW.OFF2 )
   END_RUNG
   RUNG wire#w1
      R_Coil( #Output.ACT.CW.OFF3 )
   END_RUNG
   RUNG wire#w1
      R_Coil( #Output.ACT.CW.INHIBIT_OPREATION )
   END_RUNG
   RUNG wire#w1
      R_Coil( #Output.ACT.CW.RAMP_OUT_ZERO )
   END_RUNG
   RUNG wire#w1
      R_Coil( #Output.ACT.CW.RAMP_HOLD )
   END_RUNG
   RUNG wire#w1
      R_Coil( #Output.ACT.CW.RAMP_IN_ZERO )
   END_RUNG
   RUNG wire#w1
      { S7_GenerateENO := "TRUE" } Move(in := 10, out1 => #POWER_STATE)
      wire#w2
      Coil( #STOPPED )
   END_RUNG
   RUNG wire#w2
      Not()
      Coil( #RUNNING )
   END_RUNG
   // the same network as SCL:
   // ENO of a box is taken as its EN; it also drops when the box reports an error
   #_w1 := (#POWER_STATE = 3) OR (#POWER_STATE = 5);
   IF #_w1 THEN
       #Output.ACT.CW.OFF1 := FALSE;
       #Output.ACT.CW.OFF2 := FALSE;
       #Output.ACT.CW.OFF3 := FALSE;
       #Output.ACT.CW.INHIBIT_OPREATION := FALSE;
       #Output.ACT.CW.RAMP_OUT_ZERO := FALSE;
       #Output.ACT.CW.RAMP_HOLD := FALSE;
       #Output.ACT.CW.RAMP_IN_ZERO := FALSE;
       #POWER_STATE := 10;
   END_IF;
   #STOPPED := #_w1;
   #RUNNING := NOT #_w1;
END_REGION

REGION Network 35: Switch on
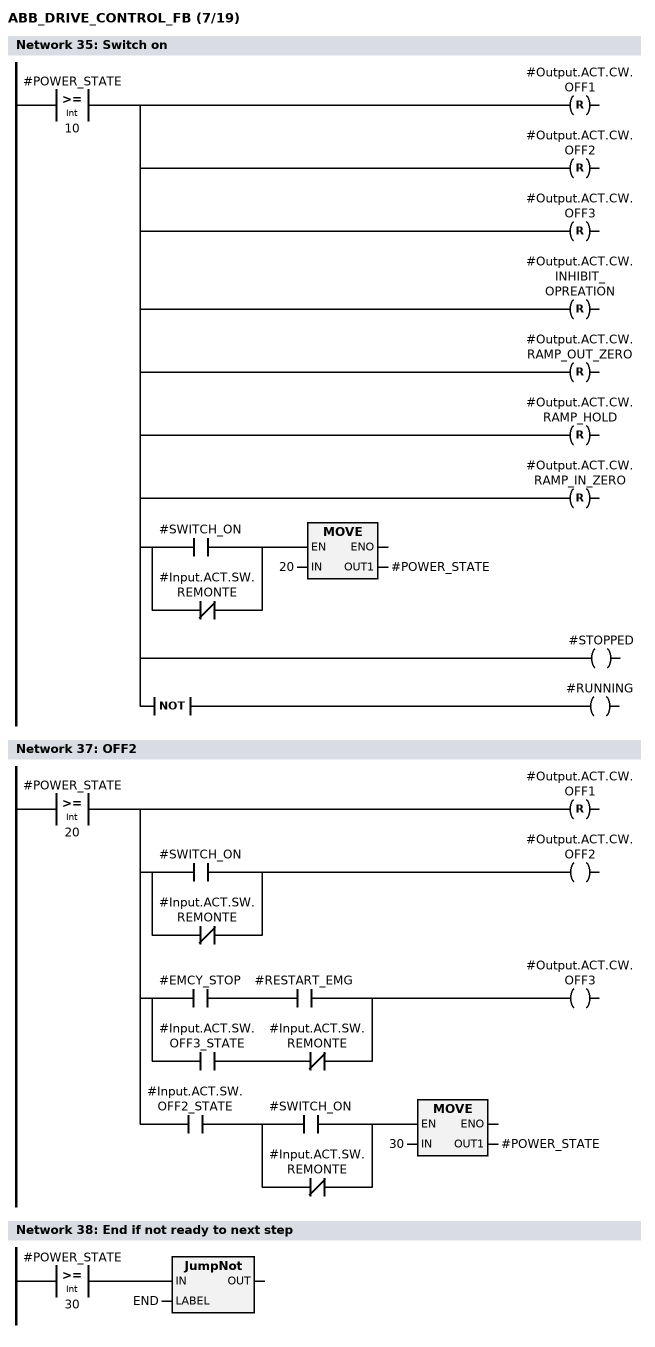
   RUNG wire#powerrail
      { S7_Templates := "SrcType := Int" } GE_Contact(in1 := #POWER_STATE, in2 := 10)
      wire#w1
      R_Coil( #Output.ACT.CW.OFF1 )
   END_RUNG
   RUNG wire#w1
      R_Coil( #Output.ACT.CW.OFF2 )
   END_RUNG
   RUNG wire#w1
      R_Coil( #Output.ACT.CW.OFF3 )
   END_RUNG
   RUNG wire#w1
      R_Coil( #Output.ACT.CW.INHIBIT_OPREATION )
   END_RUNG
   RUNG wire#w1
      R_Coil( #Output.ACT.CW.RAMP_OUT_ZERO )
   END_RUNG
   RUNG wire#w1
      R_Coil( #Output.ACT.CW.RAMP_HOLD )
   END_RUNG
   RUNG wire#w1
      R_Coil( #Output.ACT.CW.RAMP_IN_ZERO )
   END_RUNG
   RUNG wire#w1
      Contact( #SWITCH_ON )
      wire#w2
      { S7_GenerateENO := "TRUE" } Move(in := 20, out1 => #POWER_STATE)
   END_RUNG
   RUNG wire#w1
      I_Contact( #Input.ACT.SW.REMONTE )
   END_RUNG wire#w2
   RUNG wire#w1
      Coil( #STOPPED )
   END_RUNG
   RUNG wire#w1
      Not()
      Coil( #RUNNING )
   END_RUNG
   // the same network as SCL:
   #_w1 := #POWER_STATE >= 10;
   IF #_w1 THEN
       #Output.ACT.CW.OFF1 := FALSE;
       #Output.ACT.CW.OFF2 := FALSE;
       #Output.ACT.CW.OFF3 := FALSE;
       #Output.ACT.CW.INHIBIT_OPREATION := FALSE;
       #Output.ACT.CW.RAMP_OUT_ZERO := FALSE;
       #Output.ACT.CW.RAMP_HOLD := FALSE;
       #Output.ACT.CW.RAMP_IN_ZERO := FALSE;
   END_IF;
   IF #_w1 AND (#SWITCH_ON OR NOT #Input.ACT.SW.REMONTE) THEN #POWER_STATE := 20; END_IF;
   #STOPPED := #_w1;
   #RUNNING := NOT #_w1;
END_REGION

REGION Network 36: Future use
END_REGION

REGION Network 37: OFF2
   RUNG wire#powerrail
      { S7_Templates := "SrcType := Int" } GE_Contact(in1 := #POWER_STATE, in2 := 20)
      wire#w1
      R_Coil( #Output.ACT.CW.OFF1 )
   END_RUNG
   RUNG wire#w1
      Contact( #SWITCH_ON )
      wire#w2
      Coil( #Output.ACT.CW.OFF2 )
   END_RUNG
   RUNG wire#w1
      I_Contact( #Input.ACT.SW.REMONTE )
   END_RUNG wire#w2
   RUNG wire#w1
      Contact( #EMCY_STOP )
      Contact( #RESTART_EMG )
      wire#w3
      Coil( #Output.ACT.CW.OFF3 )
   END_RUNG
   RUNG wire#w1
      Contact( #Input.ACT.SW.OFF3_STATE )
      I_Contact( #Input.ACT.SW.REMONTE )
   END_RUNG wire#w3
   RUNG wire#w1
      Contact( #Input.ACT.SW.OFF2_STATE )
      wire#w4
      Contact( #SWITCH_ON )
      wire#w5
      { S7_GenerateENO := "TRUE" } Move(in := 30, out1 => #POWER_STATE)
   END_RUNG
   RUNG wire#w4
      I_Contact( #Input.ACT.SW.REMONTE )
   END_RUNG wire#w5
   // the same network as SCL:
   #_w1 := #POWER_STATE >= 20;
   IF #_w1 THEN #Output.ACT.CW.OFF1 := FALSE; END_IF;
   #Output.ACT.CW.OFF2 := #_w1 AND (#SWITCH_ON OR NOT #Input.ACT.SW.REMONTE);
   #Output.ACT.CW.OFF3 := #_w1 AND ((#EMCY_STOP AND #RESTART_EMG) OR (#Input.ACT.SW.OFF3_STATE AND NOT #Input.ACT.SW.REMONTE));
   IF #_w1 AND #Input.ACT.SW.OFF2_STATE AND (#SWITCH_ON OR NOT #Input.ACT.SW.REMONTE) THEN
       #POWER_STATE := 30;
   END_IF;
END_REGION

REGION Network 38: End if not ready to next step
   // no SCL statement known for JumpNot: written as a call
   JumpNot(in := #POWER_STATE >= 30, label := END);
END_REGION

REGION Network 39: OFF3
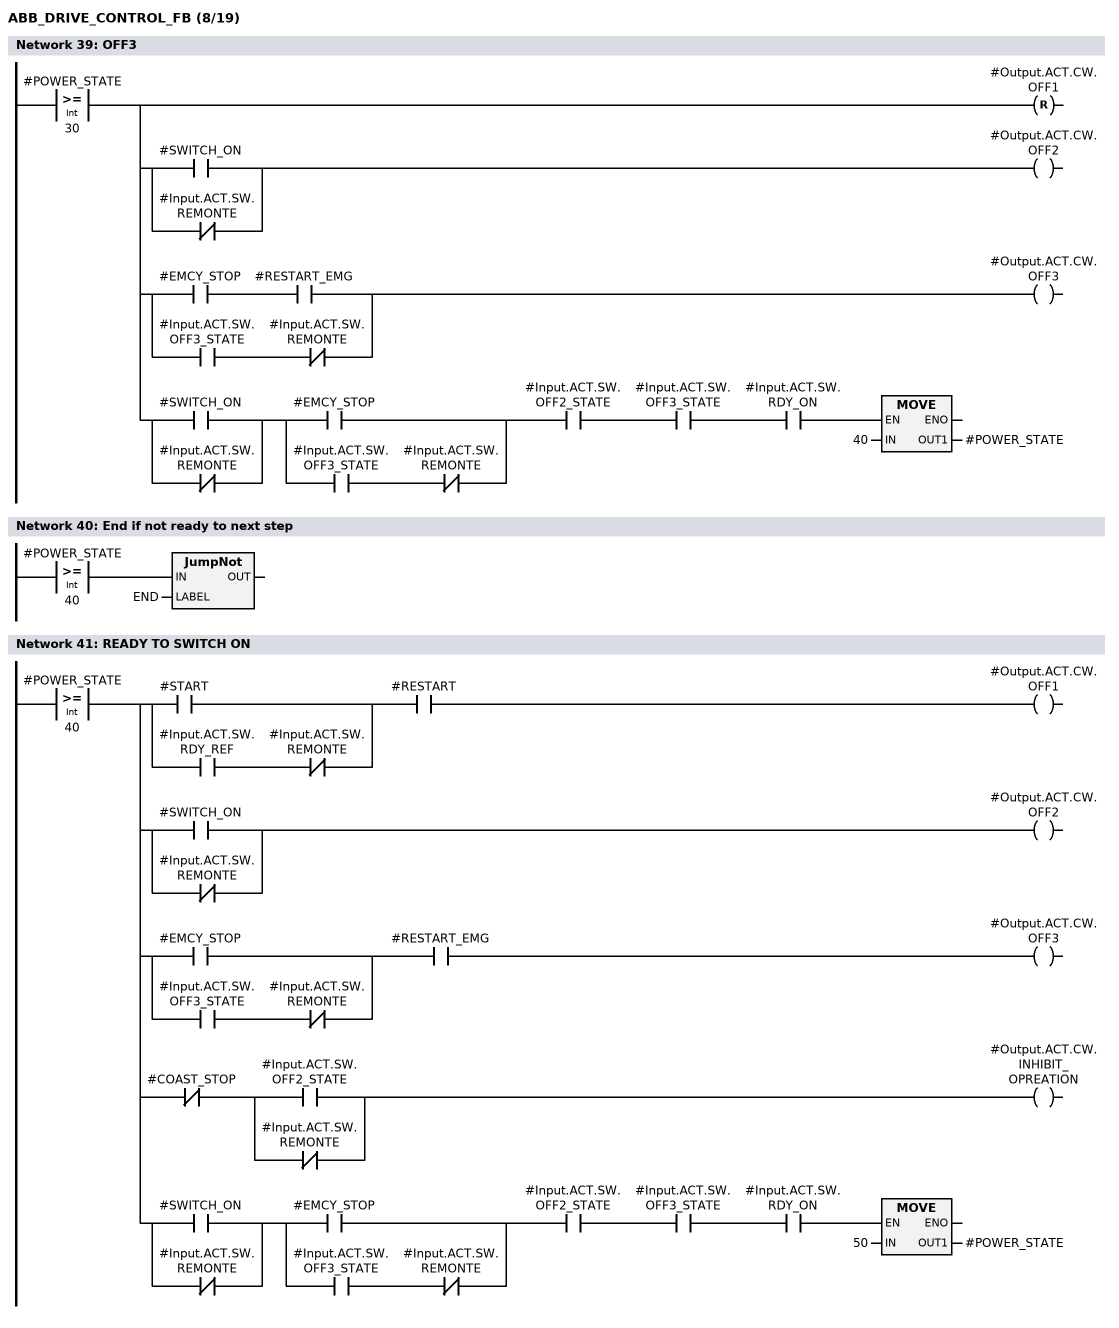
   RUNG wire#powerrail
      { S7_Templates := "SrcType := Int" } GE_Contact(in1 := #POWER_STATE, in2 := 30)
      wire#w1
      R_Coil( #Output.ACT.CW.OFF1 )
   END_RUNG
   RUNG wire#w1
      Contact( #SWITCH_ON )
      wire#w2
      Coil( #Output.ACT.CW.OFF2 )
   END_RUNG
   RUNG wire#w1
      I_Contact( #Input.ACT.SW.REMONTE )
   END_RUNG wire#w2
   RUNG wire#w1
      Contact( #EMCY_STOP )
      Contact( #RESTART_EMG )
      wire#w3
      Coil( #Output.ACT.CW.OFF3 )
   END_RUNG
   RUNG wire#w1
      Contact( #Input.ACT.SW.OFF3_STATE )
      I_Contact( #Input.ACT.SW.REMONTE )
   END_RUNG wire#w3
   RUNG wire#w1
      Contact( #SWITCH_ON )
      wire#w4
      Contact( #EMCY_STOP )
      wire#w5
      Contact( #Input.ACT.SW.OFF2_STATE )
      Contact( #Input.ACT.SW.OFF3_STATE )
      Contact( #Input.ACT.SW.RDY_ON )
      { S7_GenerateENO := "TRUE" } Move(in := 40, out1 => #POWER_STATE)
   END_RUNG
   RUNG wire#w1
      I_Contact( #Input.ACT.SW.REMONTE )
   END_RUNG wire#w4
   RUNG wire#w4
      Contact( #Input.ACT.SW.OFF3_STATE )
      I_Contact( #Input.ACT.SW.REMONTE )
   END_RUNG wire#w5
   // the same network as SCL:
   #_w1 := #POWER_STATE >= 30;
   IF #_w1 THEN #Output.ACT.CW.OFF1 := FALSE; END_IF;
   #Output.ACT.CW.OFF2 := #_w1 AND (#SWITCH_ON OR NOT #Input.ACT.SW.REMONTE);
   #Output.ACT.CW.OFF3 := #_w1 AND ((#EMCY_STOP AND #RESTART_EMG) OR (#Input.ACT.SW.OFF3_STATE AND NOT #Input.ACT.SW.REMONTE));
   IF #_w1 AND (#SWITCH_ON OR NOT #Input.ACT.SW.REMONTE) AND (#EMCY_STOP OR (#Input.ACT.SW.OFF3_STATE AND NOT #Input.ACT.SW.REMONTE)) AND #Input.ACT.SW.OFF2_STATE AND #Input.ACT.SW.OFF3_STATE AND #Input.ACT.SW.RDY_ON THEN
       #POWER_STATE := 40;
   END_IF;
END_REGION

REGION Network 40: End if not ready to next step
   // no SCL statement known for JumpNot: written as a call
   JumpNot(in := #POWER_STATE >= 40, label := END);
END_REGION

REGION Network 41: READY TO SWITCH ON
   RUNG wire#powerrail
      { S7_Templates := "SrcType := Int" } GE_Contact(in1 := #POWER_STATE, in2 := 40)
      wire#w1
      Contact( #START )
      wire#w2
      Contact( #RESTART )
      Coil( #Output.ACT.CW.OFF1 )
   END_RUNG
   RUNG wire#w1
      Contact( #Input.ACT.SW.RDY_REF )
      I_Contact( #Input.ACT.SW.REMONTE )
   END_RUNG wire#w2
   RUNG wire#w1
      Contact( #SWITCH_ON )
      wire#w3
      Coil( #Output.ACT.CW.OFF2 )
   END_RUNG
   RUNG wire#w1
      I_Contact( #Input.ACT.SW.REMONTE )
   END_RUNG wire#w3
   RUNG wire#w1
      Contact( #EMCY_STOP )
      wire#w4
      Contact( #RESTART_EMG )
      Coil( #Output.ACT.CW.OFF3 )
   END_RUNG
   RUNG wire#w1
      Contact( #Input.ACT.SW.OFF3_STATE )
      I_Contact( #Input.ACT.SW.REMONTE )
   END_RUNG wire#w4
   RUNG wire#w1
      I_Contact( #COAST_STOP )
      wire#w5
      Contact( #Input.ACT.SW.OFF2_STATE )
      wire#w6
      Coil( #Output.ACT.CW.INHIBIT_OPREATION )
   END_RUNG
   RUNG wire#w5
      I_Contact( #Input.ACT.SW.REMONTE )
   END_RUNG wire#w6
   RUNG wire#w1
      Contact( #SWITCH_ON )
      wire#w7
      Contact( #EMCY_STOP )
      wire#w8
      Contact( #Input.ACT.SW.OFF2_STATE )
      Contact( #Input.ACT.SW.OFF3_STATE )
      Contact( #Input.ACT.SW.RDY_ON )
      { S7_GenerateENO := "TRUE" } Move(in := 50, out1 => #POWER_STATE)
   END_RUNG
   RUNG wire#w1
      I_Contact( #Input.ACT.SW.REMONTE )
   END_RUNG wire#w7
   RUNG wire#w7
      Contact( #Input.ACT.SW.OFF3_STATE )
      I_Contact( #Input.ACT.SW.REMONTE )
   END_RUNG wire#w8
   // the same network as SCL:
   #_w1 := #POWER_STATE >= 40;
   #Output.ACT.CW.OFF1 := #_w1 AND (#START OR (#Input.ACT.SW.RDY_REF AND NOT #Input.ACT.SW.REMONTE)) AND #RESTART;
   #Output.ACT.CW.OFF2 := #_w1 AND (#SWITCH_ON OR NOT #Input.ACT.SW.REMONTE);
   #Output.ACT.CW.OFF3 := #_w1 AND (#EMCY_STOP OR (#Input.ACT.SW.OFF3_STATE AND NOT #Input.ACT.SW.REMONTE)) AND #RESTART_EMG;
   #Output.ACT.CW.INHIBIT_OPREATION := #_w1 AND NOT #COAST_STOP AND (#Input.ACT.SW.OFF2_STATE OR NOT #Input.ACT.SW.REMONTE);
   IF #_w1 AND (#SWITCH_ON OR NOT #Input.ACT.SW.REMONTE) AND (#EMCY_STOP OR (#Input.ACT.SW.OFF3_STATE AND NOT #Input.ACT.SW.REMONTE)) AND #Input.ACT.SW.OFF2_STATE AND #Input.ACT.SW.OFF3_STATE AND #Input.ACT.SW.RDY_ON THEN
       #POWER_STATE := 50;
   END_IF;
END_REGION

REGION Network 42: End if not ready to next step
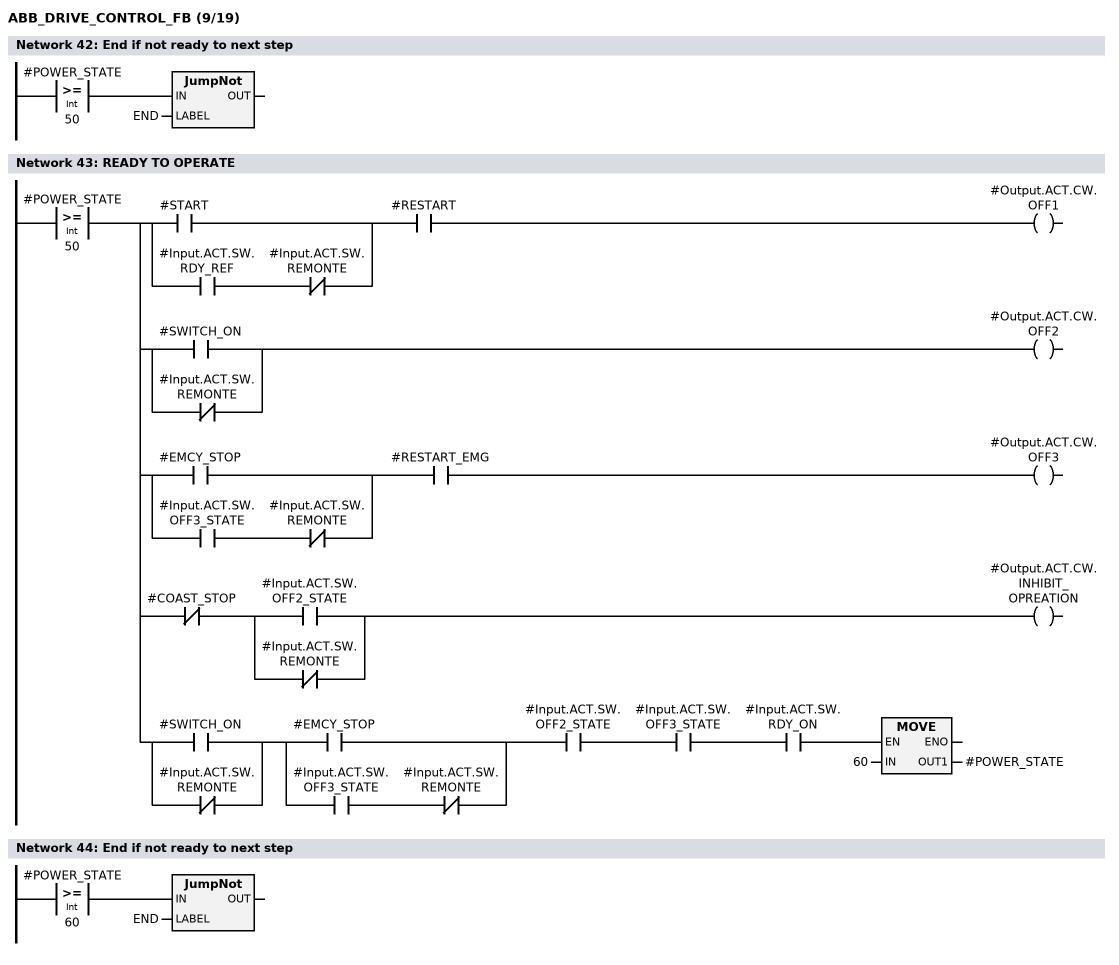
   // no SCL statement known for JumpNot: written as a call
   JumpNot(in := #POWER_STATE >= 50, label := END);
END_REGION

REGION Network 43: READY TO OPERATE
   RUNG wire#powerrail
      { S7_Templates := "SrcType := Int" } GE_Contact(in1 := #POWER_STATE, in2 := 50)
      wire#w1
      Contact( #START )
      wire#w2
      Contact( #RESTART )
      Coil( #Output.ACT.CW.OFF1 )
   END_RUNG
   RUNG wire#w1
      Contact( #Input.ACT.SW.RDY_REF )
      I_Contact( #Input.ACT.SW.REMONTE )
   END_RUNG wire#w2
   RUNG wire#w1
      Contact( #SWITCH_ON )
      wire#w3
      Coil( #Output.ACT.CW.OFF2 )
   END_RUNG
   RUNG wire#w1
      I_Contact( #Input.ACT.SW.REMONTE )
   END_RUNG wire#w3
   RUNG wire#w1
      Contact( #EMCY_STOP )
      wire#w4
      Contact( #RESTART_EMG )
      Coil( #Output.ACT.CW.OFF3 )
   END_RUNG
   RUNG wire#w1
      Contact( #Input.ACT.SW.OFF3_STATE )
      I_Contact( #Input.ACT.SW.REMONTE )
   END_RUNG wire#w4
   RUNG wire#w1
      I_Contact( #COAST_STOP )
      wire#w5
      Contact( #Input.ACT.SW.OFF2_STATE )
      wire#w6
      Coil( #Output.ACT.CW.INHIBIT_OPREATION )
   END_RUNG
   RUNG wire#w5
      I_Contact( #Input.ACT.SW.REMONTE )
   END_RUNG wire#w6
   RUNG wire#w1
      Contact( #SWITCH_ON )
      wire#w7
      Contact( #EMCY_STOP )
      wire#w8
      Contact( #Input.ACT.SW.OFF2_STATE )
      Contact( #Input.ACT.SW.OFF3_STATE )
      Contact( #Input.ACT.SW.RDY_ON )
      { S7_GenerateENO := "TRUE" } Move(in := 60, out1 => #POWER_STATE)
   END_RUNG
   RUNG wire#w1
      I_Contact( #Input.ACT.SW.REMONTE )
   END_RUNG wire#w7
   RUNG wire#w7
      Contact( #Input.ACT.SW.OFF3_STATE )
      I_Contact( #Input.ACT.SW.REMONTE )
   END_RUNG wire#w8
   // the same network as SCL:
   #_w1 := #POWER_STATE >= 50;
   #Output.ACT.CW.OFF1 := #_w1 AND (#START OR (#Input.ACT.SW.RDY_REF AND NOT #Input.ACT.SW.REMONTE)) AND #RESTART;
   #Output.ACT.CW.OFF2 := #_w1 AND (#SWITCH_ON OR NOT #Input.ACT.SW.REMONTE);
   #Output.ACT.CW.OFF3 := #_w1 AND (#EMCY_STOP OR (#Input.ACT.SW.OFF3_STATE AND NOT #Input.ACT.SW.REMONTE)) AND #RESTART_EMG;
   #Output.ACT.CW.INHIBIT_OPREATION := #_w1 AND NOT #COAST_STOP AND (#Input.ACT.SW.OFF2_STATE OR NOT #Input.ACT.SW.REMONTE);
   IF #_w1 AND (#SWITCH_ON OR NOT #Input.ACT.SW.REMONTE) AND (#EMCY_STOP OR (#Input.ACT.SW.OFF3_STATE AND NOT #Input.ACT.SW.REMONTE)) AND #Input.ACT.SW.OFF2_STATE AND #Input.ACT.SW.OFF3_STATE AND #Input.ACT.SW.RDY_ON THEN
       #POWER_STATE := 60;
   END_IF;
END_REGION

REGION Network 44: End if not ready to next step
   // no SCL statement known for JumpNot: written as a call
   JumpNot(in := #POWER_STATE >= 60, label := END);
END_REGION

REGION Network 45: OPERATION ENABLE
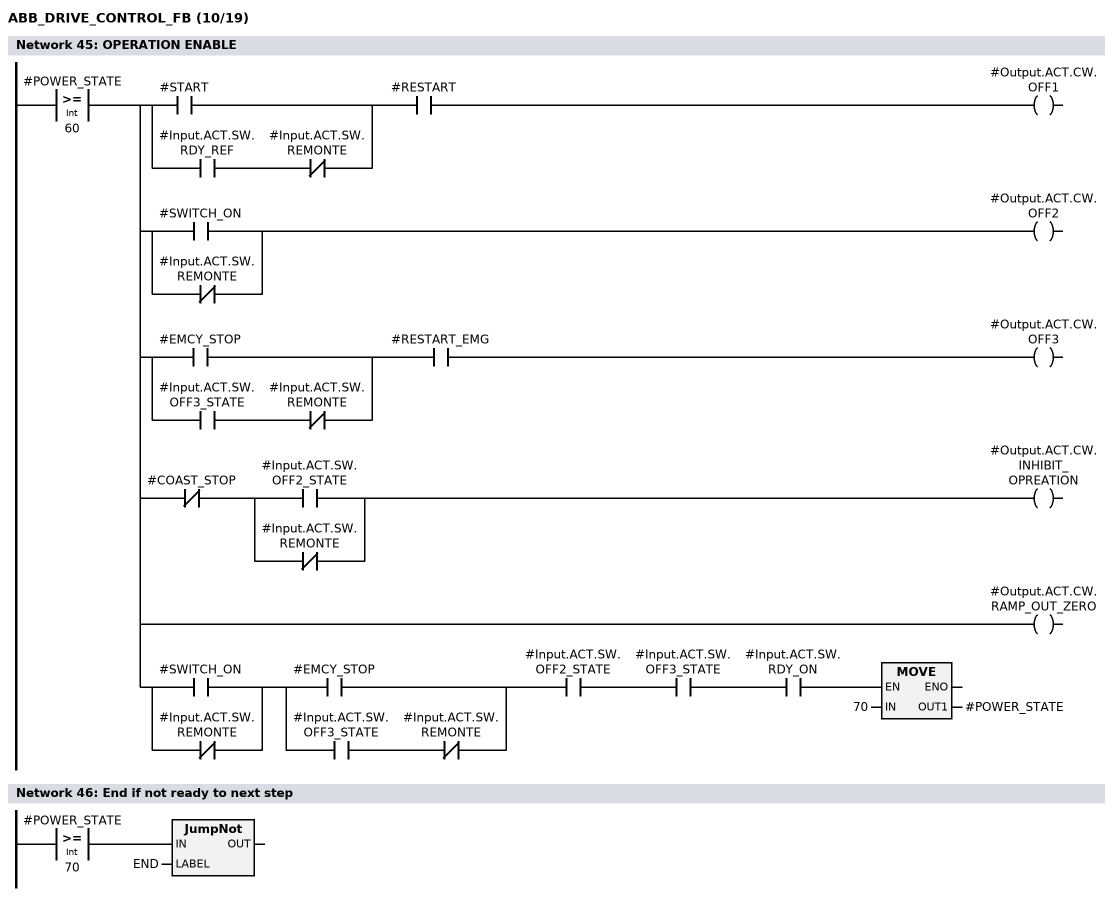
   RUNG wire#powerrail
      { S7_Templates := "SrcType := Int" } GE_Contact(in1 := #POWER_STATE, in2 := 60)
      wire#w1
      Contact( #START )
      wire#w2
      Contact( #RESTART )
      Coil( #Output.ACT.CW.OFF1 )
   END_RUNG
   RUNG wire#w1
      Contact( #Input.ACT.SW.RDY_REF )
      I_Contact( #Input.ACT.SW.REMONTE )
   END_RUNG wire#w2
   RUNG wire#w1
      Contact( #SWITCH_ON )
      wire#w3
      Coil( #Output.ACT.CW.OFF2 )
   END_RUNG
   RUNG wire#w1
      I_Contact( #Input.ACT.SW.REMONTE )
   END_RUNG wire#w3
   RUNG wire#w1
      Contact( #EMCY_STOP )
      wire#w4
      Contact( #RESTART_EMG )
      Coil( #Output.ACT.CW.OFF3 )
   END_RUNG
   RUNG wire#w1
      Contact( #Input.ACT.SW.OFF3_STATE )
      I_Contact( #Input.ACT.SW.REMONTE )
   END_RUNG wire#w4
   RUNG wire#w1
      I_Contact( #COAST_STOP )
      wire#w5
      Contact( #Input.ACT.SW.OFF2_STATE )
      wire#w6
      Coil( #Output.ACT.CW.INHIBIT_OPREATION )
   END_RUNG
   RUNG wire#w5
      I_Contact( #Input.ACT.SW.REMONTE )
   END_RUNG wire#w6
   RUNG wire#w1
      Coil( #Output.ACT.CW.RAMP_OUT_ZERO )
   END_RUNG
   RUNG wire#w1
      Contact( #SWITCH_ON )
      wire#w7
      Contact( #EMCY_STOP )
      wire#w8
      Contact( #Input.ACT.SW.OFF2_STATE )
      Contact( #Input.ACT.SW.OFF3_STATE )
      Contact( #Input.ACT.SW.RDY_ON )
      { S7_GenerateENO := "TRUE" } Move(in := 70, out1 => #POWER_STATE)
   END_RUNG
   RUNG wire#w1
      I_Contact( #Input.ACT.SW.REMONTE )
   END_RUNG wire#w7
   RUNG wire#w7
      Contact( #Input.ACT.SW.OFF3_STATE )
      I_Contact( #Input.ACT.SW.REMONTE )
   END_RUNG wire#w8
   // the same network as SCL:
   #_w1 := #POWER_STATE >= 60;
   #Output.ACT.CW.OFF1 := #_w1 AND (#START OR (#Input.ACT.SW.RDY_REF AND NOT #Input.ACT.SW.REMONTE)) AND #RESTART;
   #Output.ACT.CW.OFF2 := #_w1 AND (#SWITCH_ON OR NOT #Input.ACT.SW.REMONTE);
   #Output.ACT.CW.OFF3 := #_w1 AND (#EMCY_STOP OR (#Input.ACT.SW.OFF3_STATE AND NOT #Input.ACT.SW.REMONTE)) AND #RESTART_EMG;
   #Output.ACT.CW.INHIBIT_OPREATION := #_w1 AND NOT #COAST_STOP AND (#Input.ACT.SW.OFF2_STATE OR NOT #Input.ACT.SW.REMONTE);
   #Output.ACT.CW.RAMP_OUT_ZERO := #_w1;
   IF #_w1 AND (#SWITCH_ON OR NOT #Input.ACT.SW.REMONTE) AND (#EMCY_STOP OR (#Input.ACT.SW.OFF3_STATE AND NOT #Input.ACT.SW.REMONTE)) AND #Input.ACT.SW.OFF2_STATE AND #Input.ACT.SW.OFF3_STATE AND #Input.ACT.SW.RDY_ON THEN
       #POWER_STATE := 70;
   END_IF;
END_REGION

REGION Network 46: End if not ready to next step
   // no SCL statement known for JumpNot: written as a call
   JumpNot(in := #POWER_STATE >= 70, label := END);
END_REGION

REGION Network 47: SET RAMP HOLD
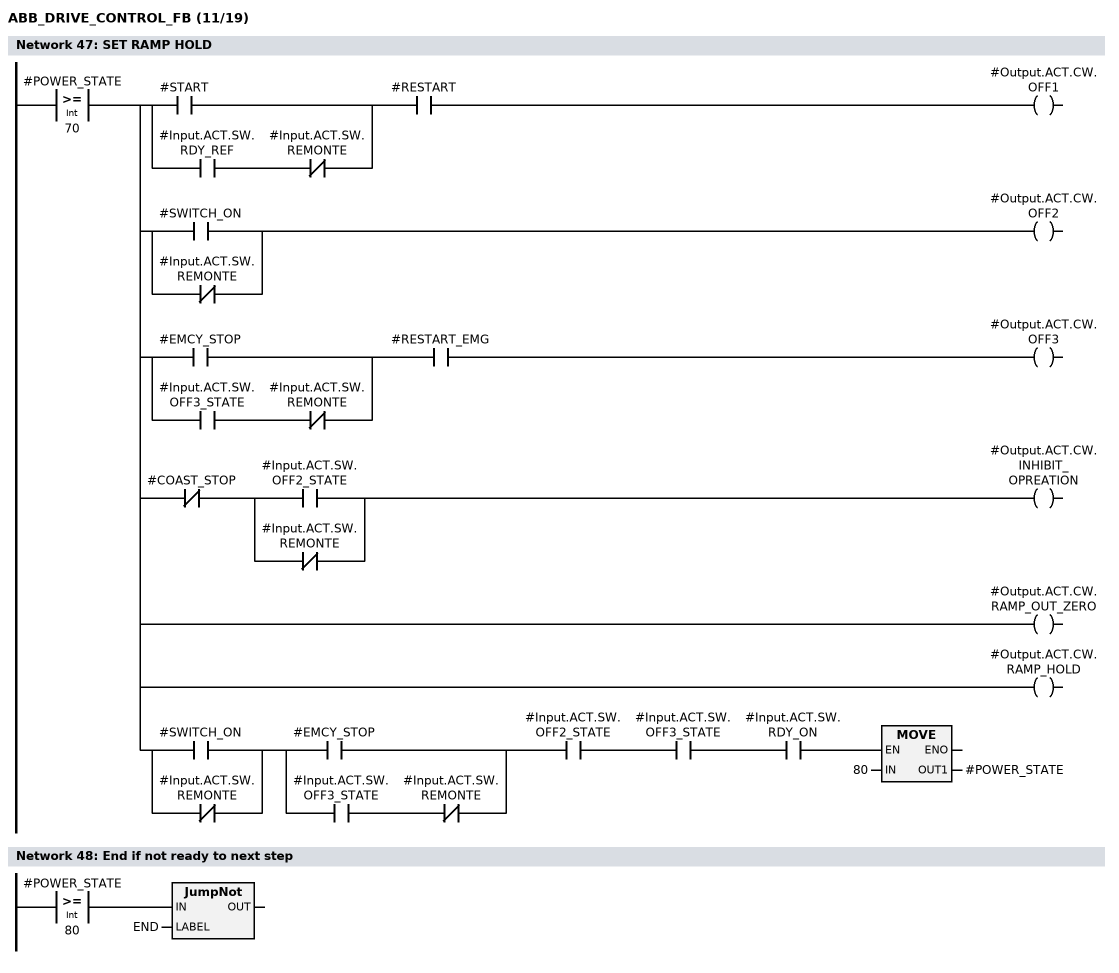
   RUNG wire#powerrail
      { S7_Templates := "SrcType := Int" } GE_Contact(in1 := #POWER_STATE, in2 := 70)
      wire#w1
      Contact( #START )
      wire#w2
      Contact( #RESTART )
      Coil( #Output.ACT.CW.OFF1 )
   END_RUNG
   RUNG wire#w1
      Contact( #Input.ACT.SW.RDY_REF )
      I_Contact( #Input.ACT.SW.REMONTE )
   END_RUNG wire#w2
   RUNG wire#w1
      Contact( #SWITCH_ON )
      wire#w3
      Coil( #Output.ACT.CW.OFF2 )
   END_RUNG
   RUNG wire#w1
      I_Contact( #Input.ACT.SW.REMONTE )
   END_RUNG wire#w3
   RUNG wire#w1
      Contact( #EMCY_STOP )
      wire#w4
      Contact( #RESTART_EMG )
      Coil( #Output.ACT.CW.OFF3 )
   END_RUNG
   RUNG wire#w1
      Contact( #Input.ACT.SW.OFF3_STATE )
      I_Contact( #Input.ACT.SW.REMONTE )
   END_RUNG wire#w4
   RUNG wire#w1
      I_Contact( #COAST_STOP )
      wire#w5
      Contact( #Input.ACT.SW.OFF2_STATE )
      wire#w6
      Coil( #Output.ACT.CW.INHIBIT_OPREATION )
   END_RUNG
   RUNG wire#w5
      I_Contact( #Input.ACT.SW.REMONTE )
   END_RUNG wire#w6
   RUNG wire#w1
      Coil( #Output.ACT.CW.RAMP_OUT_ZERO )
   END_RUNG
   RUNG wire#w1
      Coil( #Output.ACT.CW.RAMP_HOLD )
   END_RUNG
   RUNG wire#w1
      Contact( #SWITCH_ON )
      wire#w7
      Contact( #EMCY_STOP )
      wire#w8
      Contact( #Input.ACT.SW.OFF2_STATE )
      Contact( #Input.ACT.SW.OFF3_STATE )
      Contact( #Input.ACT.SW.RDY_ON )
      { S7_GenerateENO := "TRUE" } Move(in := 80, out1 => #POWER_STATE)
   END_RUNG
   RUNG wire#w1
      I_Contact( #Input.ACT.SW.REMONTE )
   END_RUNG wire#w7
   RUNG wire#w7
      Contact( #Input.ACT.SW.OFF3_STATE )
      I_Contact( #Input.ACT.SW.REMONTE )
   END_RUNG wire#w8
   // the same network as SCL:
   #_w1 := #POWER_STATE >= 70;
   #Output.ACT.CW.OFF1 := #_w1 AND (#START OR (#Input.ACT.SW.RDY_REF AND NOT #Input.ACT.SW.REMONTE)) AND #RESTART;
   #Output.ACT.CW.OFF2 := #_w1 AND (#SWITCH_ON OR NOT #Input.ACT.SW.REMONTE);
   #Output.ACT.CW.OFF3 := #_w1 AND (#EMCY_STOP OR (#Input.ACT.SW.OFF3_STATE AND NOT #Input.ACT.SW.REMONTE)) AND #RESTART_EMG;
   #Output.ACT.CW.INHIBIT_OPREATION := #_w1 AND NOT #COAST_STOP AND (#Input.ACT.SW.OFF2_STATE OR NOT #Input.ACT.SW.REMONTE);
   #Output.ACT.CW.RAMP_OUT_ZERO := #_w1;
   #Output.ACT.CW.RAMP_HOLD := #_w1;
   IF #_w1 AND (#SWITCH_ON OR NOT #Input.ACT.SW.REMONTE) AND (#EMCY_STOP OR (#Input.ACT.SW.OFF3_STATE AND NOT #Input.ACT.SW.REMONTE)) AND #Input.ACT.SW.OFF2_STATE AND #Input.ACT.SW.OFF3_STATE AND #Input.ACT.SW.RDY_ON THEN
       #POWER_STATE := 80;
   END_IF;
END_REGION

REGION Network 48: End if not ready to next step
   // no SCL statement known for JumpNot: written as a call
   JumpNot(in := #POWER_STATE >= 80, label := END);
END_REGION

REGION Network 49: SET RAMP IN
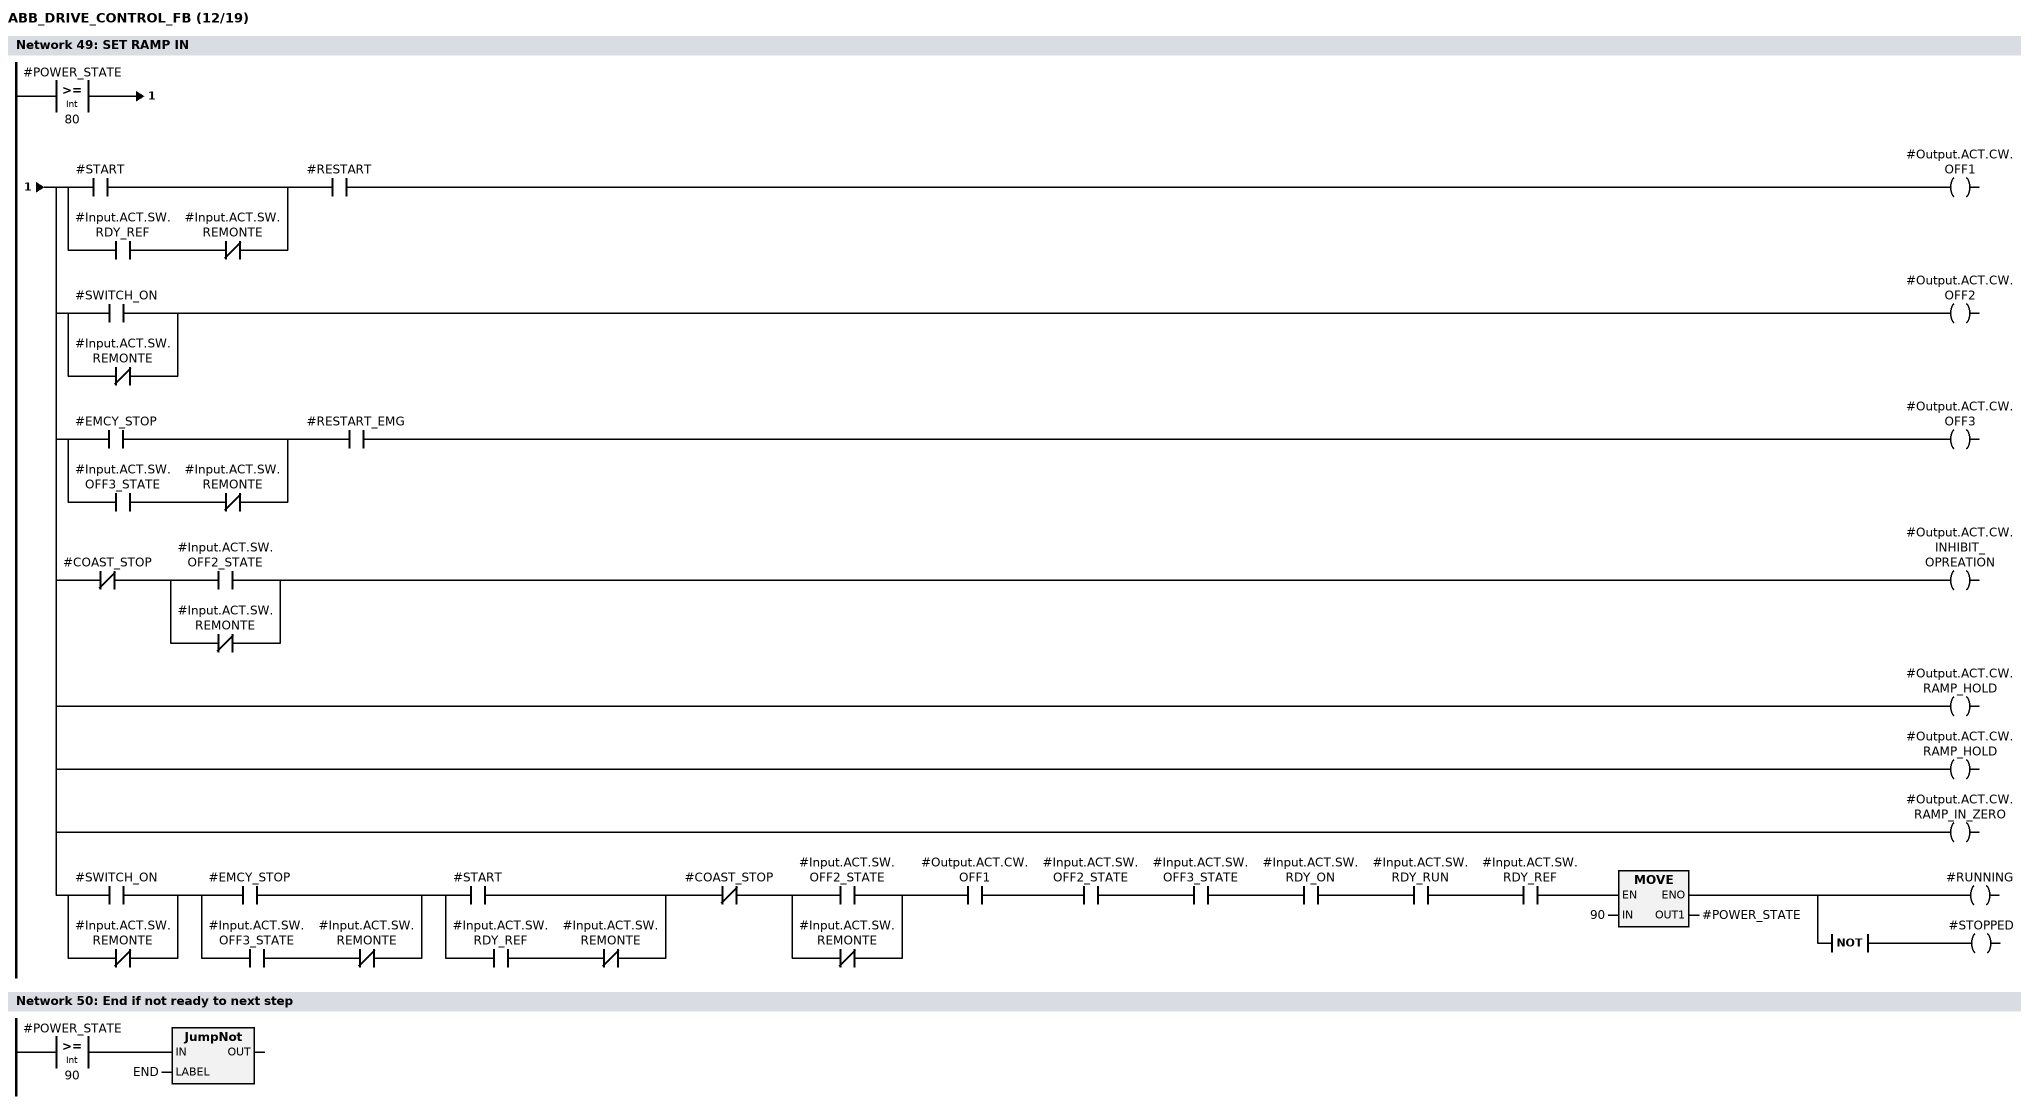
   RUNG wire#powerrail
      { S7_Templates := "SrcType := Int" } GE_Contact(in1 := #POWER_STATE, in2 := 80)
      wire#w1
      Contact( #START )
      wire#w2
      Contact( #RESTART )
      Coil( #Output.ACT.CW.OFF1 )
   END_RUNG
   RUNG wire#w1
      Contact( #Input.ACT.SW.RDY_REF )
      I_Contact( #Input.ACT.SW.REMONTE )
   END_RUNG wire#w2
   RUNG wire#w1
      Contact( #SWITCH_ON )
      wire#w3
      Coil( #Output.ACT.CW.OFF2 )
   END_RUNG
   RUNG wire#w1
      I_Contact( #Input.ACT.SW.REMONTE )
   END_RUNG wire#w3
   RUNG wire#w1
      Contact( #EMCY_STOP )
      wire#w4
      Contact( #RESTART_EMG )
      Coil( #Output.ACT.CW.OFF3 )
   END_RUNG
   RUNG wire#w1
      Contact( #Input.ACT.SW.OFF3_STATE )
      I_Contact( #Input.ACT.SW.REMONTE )
   END_RUNG wire#w4
   RUNG wire#w1
      I_Contact( #COAST_STOP )
      wire#w5
      Contact( #Input.ACT.SW.OFF2_STATE )
      wire#w6
      Coil( #Output.ACT.CW.INHIBIT_OPREATION )
   END_RUNG
   RUNG wire#w5
      I_Contact( #Input.ACT.SW.REMONTE )
   END_RUNG wire#w6
   RUNG wire#w1
      Coil( #Output.ACT.CW.RAMP_HOLD )
   END_RUNG
   RUNG wire#w1
      Coil( #Output.ACT.CW.RAMP_HOLD )
   END_RUNG
   RUNG wire#w1
      Coil( #Output.ACT.CW.RAMP_IN_ZERO )
   END_RUNG
   RUNG wire#w1
      Contact( #SWITCH_ON )
      wire#w7
      Contact( #EMCY_STOP )
      wire#w8
      Contact( #START )
      wire#w9
      I_Contact( #COAST_STOP )
      wire#w10
      Contact( #Input.ACT.SW.OFF2_STATE )
      wire#w11
      Contact( #Output.ACT.CW.OFF1 )
      Contact( #Input.ACT.SW.OFF2_STATE )
      Contact( #Input.ACT.SW.OFF3_STATE )
      Contact( #Input.ACT.SW.RDY_ON )
      Contact( #Input.ACT.SW.RDY_RUN )
      Contact( #Input.ACT.SW.RDY_REF )
      { S7_GenerateENO := "TRUE" } Move(in := 90, out1 => #POWER_STATE)
      wire#w12
      Coil( #RUNNING )
   END_RUNG
   RUNG wire#w1
      I_Contact( #Input.ACT.SW.REMONTE )
   END_RUNG wire#w7
   RUNG wire#w7
      Contact( #Input.ACT.SW.OFF3_STATE )
      I_Contact( #Input.ACT.SW.REMONTE )
   END_RUNG wire#w8
   RUNG wire#w8
      Contact( #Input.ACT.SW.RDY_REF )
      I_Contact( #Input.ACT.SW.REMONTE )
   END_RUNG wire#w9
   RUNG wire#w10
      I_Contact( #Input.ACT.SW.REMONTE )
   END_RUNG wire#w11
   RUNG wire#w12
      Not()
      Coil( #STOPPED )
   END_RUNG
   // the same network as SCL:
   // ENO of a box is taken as its EN; it also drops when the box reports an error
   #_w1 := #POWER_STATE >= 80;
   #Output.ACT.CW.OFF1 := #_w1 AND (#START OR (#Input.ACT.SW.RDY_REF AND NOT #Input.ACT.SW.REMONTE)) AND #RESTART;
   #Output.ACT.CW.OFF2 := #_w1 AND (#SWITCH_ON OR NOT #Input.ACT.SW.REMONTE);
   #Output.ACT.CW.OFF3 := #_w1 AND (#EMCY_STOP OR (#Input.ACT.SW.OFF3_STATE AND NOT #Input.ACT.SW.REMONTE)) AND #RESTART_EMG;
   #Output.ACT.CW.INHIBIT_OPREATION := #_w1 AND NOT #COAST_STOP AND (#Input.ACT.SW.OFF2_STATE OR NOT #Input.ACT.SW.REMONTE);
   #Output.ACT.CW.RAMP_HOLD := #_w1;
   #Output.ACT.CW.RAMP_HOLD := #_w1;
   #Output.ACT.CW.RAMP_IN_ZERO := #_w1;
   #_w2 := #_w1 AND (#SWITCH_ON OR NOT #Input.ACT.SW.REMONTE) AND (#EMCY_STOP OR (#Input.ACT.SW.OFF3_STATE AND NOT #Input.ACT.SW.REMONTE)) AND (#START OR (#Input.ACT.SW.RDY_REF AND NOT #Input.ACT.SW.REMONTE)) AND NOT #COAST_STOP AND (#Input.ACT.SW.OFF2_STATE OR NOT #Input.ACT.SW.REMONTE) AND #Output.ACT.CW.OFF1 AND #Input.ACT.SW.OFF2_STATE AND #Input.ACT.SW.OFF3_STATE AND #Input.ACT.SW.RDY_ON AND #Input.ACT.SW.RDY_RUN AND #Input.ACT.SW.RDY_REF;
   IF #_w2 THEN #POWER_STATE := 90; END_IF;
   #RUNNING := #_w2;
   #STOPPED := NOT #_w2;
END_REGION

